SPLINE
SPL {X   -93.623, Y  +806.710, Z    +0.000, E1   -55.511, E3 +129906.770}
SPL {X  -138.493, Y  +759.115, Z    +0.000, E1   -50.023, E3 +129954.598}
SPL {X  -149.871, Y  +737.133, Z    +0.000, E1   -43.112, E3 +129960.012}
SPL {X  -157.876, Y  +713.320, Z    +0.000, E1   -31.448, E3 +129959.788}
SPL {X  -161.323, Y  +695.531, Z    +0.000, E1   -20.168, E3 +129961.831}
SPL {X  -162.626, Y  +681.447, Z    +0.000, E1    -9.120, E3 +129961.820}
SPL {X  -162.820, Y  +671.283, Z    +0.000, E1    +0.049, E3 +129961.332}
SPL {X  -162.820, Y  +665.565, Z    +0.000, E1   +11.206, E3 +129960.995}
SPL {X  -162.820, Y  +658.993, Z    +0.000, E1   +25.845, E3 +129961.066}
SPL {X  -162.820, Y  +652.443, Z    +0.000, E1   +38.206, E3 +129961.801}
SPL {X  -162.820, Y  +640.832, Z    +0.000, E1   +55.385, E3 +129960.515}
SPL {X  -162.820, Y  +625.562, Z    +0.000, E1   +67.658, E3 +129959.568}
SPL {X  -162.820, Y  +600.578, Z    +0.000, E1   +80.831, E3 +129951.166}
SPL {X  -162.820, Y  +567.495, Z    +0.000, E1   +70.620, E3 +129986.290}
SPL {X  -162.820, Y  +416.506, Z    +0.000, E1   +71.398, E3 +130070.636}
SPL {X  -162.820, Y  +411.010, Z    +0.000, E1   +70.614, E3 +130082.087}
SPL {X  -162.820, Y  +391.151, Z    +0.000, E1   +70.927, E3 +130093.542}
SPL {X  -159.025, Y  +345.550, Z    +0.000, E1   +73.389, E3 +130099.223}
SPL {X  -158.911, Y  +345.038, Z    +0.000, E1   +72.209, E3 +130111.381}
SPL {X  -157.738, Y  +340.137, Z    +0.000, E1   +71.006, E3 +130126.198}
SPL {X  -155.731, Y  +332.978, Z    +0.000, E1   +69.670, E3 +130142.847}
SPL {X  -154.241, Y  +328.346, Z    +0.000, E1   +68.710, E3 +130153.790}
SPL {X  -151.364, Y  +320.507, Z    +0.000, E1   +68.513, E3 +130161.416}
SPL {X  -147.865, Y  +312.336, Z    +0.000, E1   +67.945, E3 +130171.706}
SPL {X  -144.739, Y  +305.928, Z    +0.000, E1   +67.540, E3 +130179.290}
SPL {X  -141.308, Y  +299.614, Z    +0.000, E1   +67.079, E3 +130187.081}
SPL {X  -137.907, Y  +293.943, Z    +0.000, E1   +66.608, E3 +130194.059}
SPL {X  -134.802, Y  +289.183, Z    +0.000, E1   +66.143, E3 +130200.195}
SPL {X  -131.727, Y  +284.801, Z    +0.000, E1   +65.590, E3 +130206.210}
SPL {X  -128.890, Y  +281.012, Z    +0.000, E1   +65.392, E3 +130209.955}
SPL {X  -121.325, Y  +271.915, Z    +0.000, E1   +67.092, E3 +130209.521}
SPL {X   -79.997, Y  +238.687, Z    +0.000, E1   +54.340, E3 +130368.277}
ENDSPLINE

SPLINE
SPL {X  -139.099, Y  +295.872, Z    +0.000, E1   +47.860, E3 +130496.153}
SPL {X  -156.463, Y  +335.448, Z    +0.000, E1   +33.333, E3 +130506.861}
SPL {X  -161.312, Y  +358.394, Z    +0.000, E1   +19.478, E3 +130508.495}
SPL {X  -162.549, Y  +371.111, Z    +0.000, E1    +9.905, E3 +130508.555}
SPL {X  -162.818, Y  +379.769, Z    +0.000, E1    +2.607, E3 +130508.297}
SPL {X  -162.820, Y  +382.897, Z    +0.000, E1    -0.379, E3 +130507.781}
SPL {X  -162.820, Y  +387.689, Z    +0.000, E1    -9.147, E3 +130507.501}
SPL {X  -162.820, Y  +392.805, Z    +0.000, E1   -19.930, E3 +130507.474}
SPL {X  -162.820, Y  +397.742, Z    +0.000, E1   -30.068, E3 +130507.506}
SPL {X  -162.820, Y  +403.938, Z    +0.000, E1   -41.112, E3 +130507.486}
SPL {X  -162.820, Y  +415.430, Z    +0.000, E1   -55.307, E3 +130507.685}
SPL {X  -162.820, Y  +466.986, Z    +0.000, E1   -71.397, E3 +130519.444}
SPL {X  -162.820, Y  +661.594, Z    +0.000, E1   -73.988, E3 +130605.070}
ENDSPLINE

SPLINE
SPL {X  -162.820, Y  +634.363, Z    +0.000, E1   -70.793, E3 +130618.648}
ENDSPLINE

SPLINE
SPL {X  -162.820, Y  +649.777, Z    +0.000, E1   -70.953, E3 +130628.407}
SPL {X  -162.820, Y  +667.477, Z    +0.000, E1   -70.889, E3 +130641.716}
SPL {X  -162.462, Y  +684.286, Z    +0.000, E1   -70.880, E3 +130653.949}
SPL {X  -160.799, Y  +699.074, Z    +0.000, E1   -70.750, E3 +130665.813}
SPL {X  -158.733, Y  +709.754, Z    +0.000, E1   -70.504, E3 +130675.696}
SPL {X  -156.566, Y  +718.194, Z    +0.000, E1   -70.115, E3 +130685.177}
SPL {X  -153.268, Y  +728.449, Z    +0.000, E1   -69.855, E3 +130694.803}
SPL {X  -149.282, Y  +738.502, Z    +0.000, E1   -69.318, E3 +130706.323}
SPL {X  -145.460, Y  +746.655, Z    +0.000, E1   -68.995, E3 +130714.338}
SPL {X  -143.061, Y  +751.243, Z    +0.000, E1   -68.459, E3 +130721.332}
SPL {X  -139.143, Y  +758.055, Z    +0.000, E1   -68.038, E3 +130728.895}
SPL {X  -136.095, Y  +762.879, Z    +0.000, E1   -67.470, E3 +130735.529}
SPL {X  -133.055, Y  +767.344, Z    +0.000, E1   -67.024, E3 +130741.161}
SPL {X  -129.955, Y  +771.593, Z    +0.000, E1   -66.476, E3 +130746.802}
SPL {X  -125.283, Y  +777.493, Z    +0.000, E1   -66.879, E3 +130749.226}
SPL {X   -78.323, Y  +816.244, Z    +0.000, E1   -56.979, E3 +130856.322}
ENDSPLINE

SPLINE
SPL {X   -93.623, Y  +806.710, Z    +0.000, E1   -55.511, E3 +131002.008}
SPL {X  -138.493, Y  +759.115, Z    +0.000, E1   -50.023, E3 +131049.836}
SPL {X  -149.871, Y  +737.133, Z    +0.000, E1   -43.112, E3 +131055.250}
SPL {X  -157.876, Y  +713.320, Z    +0.000, E1   -31.448, E3 +131055.026}
SPL {X  -161.323, Y  +695.531, Z    +0.000, E1   -20.168, E3 +131057.069}
SPL {X  -162.626, Y  +681.447, Z    +0.000, E1    -9.120, E3 +131057.058}
SPL {X  -162.820, Y  +673.597, Z    +0.000, E1    -2.055, E3 +131057.052}
SPL {X  -162.820, Y  +671.476, Z    +0.000, E1    +0.020, E3 +131056.594}
SPL {X  -162.820, Y  +668.959, Z    +0.000, E1    +4.387, E3 +131056.315}
SPL {X  -162.820, Y  +664.344, Z    +0.000, E1   +14.120, E3 +131056.214}
SPL {X  -162.820, Y  +658.993, Z    +0.000, E1   +25.845, E3 +131056.304}
SPL {X  -162.820, Y  +652.443, Z    +0.000, E1   +38.206, E3 +131057.039}
SPL {X  -162.820, Y  +640.832, Z    +0.000, E1   +55.385, E3 +131055.753}
SPL {X  -162.820, Y  +617.334, Z    +0.000, E1   +73.158, E3 +131052.067}
SPL {X  -162.820, Y  +567.495, Z    +0.000, E1   +70.620, E3 +131081.528}
SPL {X  -162.820, Y  +416.506, Z    +0.000, E1   +71.398, E3 +131165.874}
SPL {X  -162.820, Y  +411.010, Z    +0.000, E1   +70.614, E3 +131177.325}
SPL {X  -162.820, Y  +399.588, Z    +0.000, E1   +70.462, E3 +131187.099}
SPL {X  -159.703, Y  +348.793, Z    +0.000, E1   +73.194, E3 +131194.403}
SPL {X  -158.809, Y  +344.584, Z    +0.000, E1   +72.042, E3 +131208.707}
SPL {X  -157.517, Y  +339.284, Z    +0.000, E1   +70.832, E3 +131223.408}
SPL {X  -155.731, Y  +332.978, Z    +0.000, E1   +69.670, E3 +131238.086}
SPL {X  -154.241, Y  +328.346, Z    +0.000, E1   +68.710, E3 +131249.028}
SPL {X  -151.364, Y  +320.507, Z    +0.000, E1   +68.513, E3 +131256.655}
SPL {X  -147.865, Y  +312.336, Z    +0.000, E1   +67.945, E3 +131266.944}
SPL {X  -144.739, Y  +305.928, Z    +0.000, E1   +67.540, E3 +131274.528}
SPL {X  -141.308, Y  +299.614, Z    +0.000, E1   +67.079, E3 +131282.319}
SPL {X  -137.907, Y  +293.943, Z    +0.000, E1   +66.608, E3 +131289.297}
SPL {X  -134.802, Y  +289.183, Z    +0.000, E1   +66.143, E3 +131295.433}
SPL {X  -131.727, Y  +284.801, Z    +0.000, E1   +65.590, E3 +131301.448}
SPL {X  -128.890, Y  +281.012, Z    +0.000, E1   +65.392, E3 +131305.193}
SPL {X  -121.325, Y  +271.915, Z    +0.000, E1   +67.092, E3 +131304.759}
SPL {X   -79.997, Y  +238.687, Z    +0.000, E1   +54.340, E3 +131463.515}
ENDSPLINE

SPLINE
SPL {X  -139.099, Y  +295.872, Z    +0.000, E1   +47.860, E3 +131591.391}
SPL {X  -153.884, Y  +327.303, Z    +0.000, E1   +37.422, E3 +131602.618}
SPL {X  -160.677, Y  +354.168, Z    +0.000, E1   +22.396, E3 +131603.144}
SPL {X  -162.549, Y  +371.111, Z    +0.000, E1    +9.905, E3 +131603.793}
SPL {X  -162.818, Y  +379.769, Z    +0.000, E1    +2.607, E3 +131603.535}
SPL {X  -162.820, Y  +382.500, Z    +0.000, E1    +0.000, E3 +131603.105}
SPL {X  -162.820, Y  +384.989, Z    +0.000, E1    -3.865, E3 +131602.832}
SPL {X  -162.820, Y  +391.404, Z    +0.000, E1   -16.767, E3 +131602.678}
SPL {X  -162.820, Y  +397.742, Z    +0.000, E1   -30.068, E3 +131602.744}
SPL {X  -162.820, Y  +403.938, Z    +0.000, E1   -41.112, E3 +131602.724}
SPL {X  -162.820, Y  +415.430, Z    +0.000, E1   -55.307, E3 +131602.923}
SPL {X  -162.820, Y  +466.986, Z    +0.000, E1   -71.397, E3 +131614.682}
SPL {X  -162.820, Y  +661.594, Z    +0.000, E1   -73.988, E3 +131700.309}
ENDSPLINE

SPLINE
SPL {X  -162.820, Y  +634.363, Z    +0.000, E1   -70.793, E3 +131713.886}
ENDSPLINE

SPLINE
SPL {X  -162.820, Y  +649.777, Z    +0.000, E1   -70.953, E3 +131723.645}
SPL {X  -162.820, Y  +667.477, Z    +0.000, E1   -70.889, E3 +131736.954}
SPL {X  -162.462, Y  +684.286, Z    +0.000, E1   -70.880, E3 +131749.187}
SPL {X  -160.799, Y  +699.074, Z    +0.000, E1   -70.750, E3 +131761.051}
SPL {X  -158.733, Y  +709.754, Z    +0.000, E1   -70.504, E3 +131770.934}
SPL {X  -156.566, Y  +718.194, Z    +0.000, E1   -70.115, E3 +131780.415}
SPL {X  -153.268, Y  +728.449, Z    +0.000, E1   -69.855, E3 +131790.041}
SPL {X  -150.033, Y  +736.750, Z    +0.000, E1   -69.498, E3 +131798.752}
SPL {X  -146.704, Y  +744.128, Z    +0.000, E1   -68.985, E3 +131807.875}
SPL {X  -143.061, Y  +751.243, Z    +0.000, E1   -68.459, E3 +131816.570}
SPL {X  -139.143, Y  +758.055, Z    +0.000, E1   -68.038, E3 +131824.133}
SPL {X  -136.095, Y  +762.879, Z    +0.000, E1   -67.470, E3 +131830.767}
SPL {X  -133.055, Y  +767.344, Z    +0.000, E1   -67.024, E3 +131836.399}
SPL {X  -129.955, Y  +771.593, Z    +0.000, E1   -66.476, E3 +131842.040}
SPL {X  -125.283, Y  +777.493, Z    +0.000, E1   -66.879, E3 +131844.464}
SPL {X   -78.323, Y  +816.244, Z    +0.000, E1   -56.979, E3 +131951.560}
ENDSPLINE

SPLINE
SPL {X   -93.623, Y  +806.710, Z    +0.000, E1   -55.511, E3 +132097.246}
SPL {X  -143.027, Y  +751.304, Z    +0.000, E1   -47.932, E3 +132147.307}
SPL {X  -157.876, Y  +713.320, Z    +0.000, E1   -31.448, E3 +132150.264}
SPL {X  -161.323, Y  +695.531, Z    +0.000, E1   -20.168, E3 +132152.308}
SPL {X  -162.428, Y  +684.786, Z    +0.000, E1   -11.829, E3 +132152.205}
SPL {X  -162.809, Y  +675.372, Z    +0.000, E1    -3.788, E3 +132152.319}
SPL {X  -162.820, Y  +671.476, Z    +0.000, E1    +0.020, E3 +132151.832}
SPL {X  -162.820, Y  +668.959, Z    +0.000, E1    +4.387, E3 +132151.553}
SPL {X  -162.820, Y  +664.344, Z    +0.000, E1   +14.120, E3 +132151.452}
SPL {X  -162.820, Y  +658.993, Z    +0.000, E1   +25.845, E3 +132151.542}
SPL {X  -162.820, Y  +652.443, Z    +0.000, E1   +38.206, E3 +132152.277}
SPL {X  -162.820, Y  +640.832, Z    +0.000, E1   +55.385, E3 +132150.991}
SPL {X  -162.820, Y  +625.562, Z    +0.000, E1   +67.658, E3 +132150.044}
SPL {X  -162.820, Y  +600.578, Z    +0.000, E1   +80.831, E3 +132141.642}
SPL {X  -162.820, Y  +567.495, Z    +0.000, E1   +70.620, E3 +132176.767}
SPL {X  -162.820, Y  +416.506, Z    +0.000, E1   +71.398, E3 +132261.112}
SPL {X  -162.820, Y  +411.010, Z    +0.000, E1   +70.614, E3 +132272.563}
SPL {X  -162.820, Y  +399.588, Z    +0.000, E1   +70.462, E3 +132282.337}
SPL {X  -159.703, Y  +348.793, Z    +0.000, E1   +73.194, E3 +132289.641}
SPL {X  -158.809, Y  +344.584, Z    +0.000, E1   +72.042, E3 +132303.946}
SPL {X  -157.517, Y  +339.284, Z    +0.000, E1   +70.832, E3 +132318.647}
SPL {X  -155.731, Y  +332.978, Z    +0.000, E1   +69.670, E3 +132333.324}
SPL {X  -153.052, Y  +324.954, Z    +0.000, E1   +68.671, E3 +132347.286}
SPL {X  -149.405, Y  +315.782, Z    +0.000, E1   +68.161, E3 +132358.052}
SPL {X  -145.408, Y  +307.240, Z    +0.000, E1   +67.667, E3 +132368.030}
SPL {X  -142.385, Y  +301.526, Z    +0.000, E1   +67.199, E3 +132375.262}
SPL {X  -138.888, Y  +295.526, Z    +0.000, E1   +66.767, E3 +132382.547}
SPL {X  -134.802, Y  +289.183, Z    +0.000, E1   +66.143, E3 +132390.671}
SPL {X  -131.727, Y  +284.801, Z    +0.000, E1   +65.590, E3 +132396.686}
SPL {X  -128.890, Y  +281.012, Z    +0.000, E1   +65.392, E3 +132400.431}
SPL {X  -121.325, Y  +271.915, Z    +0.000, E1   +67.092, E3 +132399.997}
SPL {X   -79.997, Y  +238.687, Z    +0.000, E1   +54.340, E3 +132558.753}
ENDSPLINE

SPLINE
SPL {X  -139.099, Y  +295.872, Z    +0.000, E1   +47.860, E3 +132686.629}
SPL {X  -156.463, Y  +335.448, Z    +0.000, E1   +33.333, E3 +132697.337}
SPL {X  -161.312, Y  +358.394, Z    +0.000, E1   +19.478, E3 +132698.972}
SPL {X  -162.549, Y  +371.111, Z    +0.000, E1    +9.905, E3 +132699.031}
SPL {X  -162.818, Y  +379.769, Z    +0.000, E1    +2.607, E3 +132698.773}
SPL {X  -162.820, Y  +382.897, Z    +0.000, E1    -0.379, E3 +132698.258}
SPL {X  -162.820, Y  +387.689, Z    +0.000, E1    -9.147, E3 +132697.977}
SPL {X  -162.820, Y  +392.805, Z    +0.000, E1   -19.930, E3 +132697.950}
SPL {X  -162.820, Y  +397.742, Z    +0.000, E1   -30.068, E3 +132697.982}
SPL {X  -162.820, Y  +403.938, Z    +0.000, E1   -41.112, E3 +132697.962}
SPL {X  -162.820, Y  +415.430, Z    +0.000, E1   -55.307, E3 +132698.161}
SPL {X  -162.820, Y  +466.986, Z    +0.000, E1   -71.397, E3 +132709.920}
SPL {X  -162.820, Y  +661.594, Z    +0.000, E1   -73.988, E3 +132795.547}
ENDSPLINE

SPLINE
SPL {X  -162.820, Y  +639.523, Z    +0.000, E1   -70.828, E3 +132812.623}
ENDSPLINE

SPLINE
SPL {X  -162.820, Y  +655.227, Z    +0.000, E1   -71.020, E3 +132822.049}
SPL {X  -162.820, Y  +667.477, Z    +0.000, E1   -70.889, E3 +132832.192}
SPL {X  -162.097, Y  +688.831, Z    +0.000, E1   -70.910, E3 +132847.563}
SPL {X  -159.319, Y  +707.081, Z    +0.000, E1   -70.563, E3 +132863.849}
SPL {X  -155.769, Y  +720.894, Z    +0.000, E1   -70.077, E3 +132878.059}
SPL {X  -150.995, Y  +734.417, Z    +0.000, E1   -69.635, E3 +132891.436}
SPL {X  -146.704, Y  +744.128, Z    +0.000, E1   -68.985, E3 +132903.113}
SPL {X  -143.061, Y  +751.243, Z    +0.000, E1   -68.459, E3 +132911.808}
SPL {X  -139.143, Y  +758.055, Z    +0.000, E1   -68.038, E3 +132919.371}
SPL {X  -136.095, Y  +762.879, Z    +0.000, E1   -67.470, E3 +132926.006}
SPL {X  -133.055, Y  +767.344, Z    +0.000, E1   -67.024, E3 +132931.637}
SPL {X  -129.955, Y  +771.593, Z    +0.000, E1   -66.476, E3 +132937.278}
SPL {X  -125.283, Y  +777.493, Z    +0.000, E1   -66.879, E3 +132939.702}
SPL {X   -78.323, Y  +816.244, Z    +0.000, E1   -56.979, E3 +133046.798}
ENDSPLINE

SPLINE
SPL {X   -93.623, Y  +806.710, Z    +0.000, E1   -55.511, E3 +133192.484}
SPL {X  -143.027, Y  +751.304, Z    +0.000, E1   -47.932, E3 +133242.545}
SPL {X  -157.876, Y  +713.320, Z    +0.000, E1   -31.448, E3 +133245.502}
SPL {X  -161.323, Y  +695.531, Z    +0.000, E1   -20.168, E3 +133247.546}
SPL {X  -162.428, Y  +684.786, Z    +0.000, E1   -11.829, E3 +133247.443}
SPL {X  -162.809, Y  +675.372, Z    +0.000, E1    -3.788, E3 +133247.557}
SPL {X  -162.820, Y  +671.476, Z    +0.000, E1    +0.020, E3 +133247.070}
SPL {X  -162.820, Y  +668.959, Z    +0.000, E1    +4.387, E3 +133246.791}
SPL {X  -162.820, Y  +664.344, Z    +0.000, E1   +14.120, E3 +133246.690}
SPL {X  -162.820, Y  +658.993, Z    +0.000, E1   +25.845, E3 +133246.780}
SPL {X  -162.820, Y  +652.443, Z    +0.000, E1   +38.206, E3 +133247.515}
SPL {X  -162.820, Y  +640.832, Z    +0.000, E1   +55.385, E3 +133246.229}
SPL {X  -162.820, Y  +617.334, Z    +0.000, E1   +73.158, E3 +133242.543}
SPL {X  -162.820, Y  +567.495, Z    +0.000, E1   +70.620, E3 +133272.005}
SPL {X  -162.820, Y  +416.506, Z    +0.000, E1   +71.398, E3 +133356.350}
SPL {X  -162.820, Y  +411.010, Z    +0.000, E1   +70.614, E3 +133367.801}
SPL {X  -162.820, Y  +391.151, Z    +0.000, E1   +70.927, E3 +133379.256}
SPL {X  -159.025, Y  +345.550, Z    +0.000, E1   +73.389, E3 +133384.937}
ENDSPLINE

SPLINE
SPL {X  -159.121, Y  +345.992, Z    +0.000, E1   +72.455, E3 +133393.904}
ENDSPLINE

SPLINE
SPL {X  -158.667, Y  +343.959, Z    +0.000, E1   +71.763, E3 +133402.012}
SPL {X  -157.517, Y  +339.284, Z    +0.000, E1   +70.832, E3 +133413.885}
SPL {X  -155.731, Y  +332.978, Z    +0.000, E1   +69.670, E3 +133428.562}
SPL {X  -154.241, Y  +328.346, Z    +0.000, E1   +68.710, E3 +133439.505}
SPL {X  -151.364, Y  +320.507, Z    +0.000, E1   +68.513, E3 +133447.131}
SPL {X  -147.865, Y  +312.336, Z    +0.000, E1   +67.945, E3 +133457.421}
SPL {X  -143.686, Y  +303.920, Z    +0.000, E1   +67.419, E3 +133467.451}
SPL {X  -138.888, Y  +295.526, Z    +0.000, E1   +66.767, E3 +133477.785}
SPL {X  -134.802, Y  +289.183, Z    +0.000, E1   +66.143, E3 +133485.909}
SPL {X  -131.727, Y  +284.801, Z    +0.000, E1   +65.590, E3 +133491.924}
SPL {X  -128.890, Y  +281.012, Z    +0.000, E1   +65.392, E3 +133495.669}
SPL {X  -121.325, Y  +271.915, Z    +0.000, E1   +67.092, E3 +133495.235}
SPL {X   -79.997, Y  +238.687, Z    +0.000, E1   +54.340, E3 +133653.991}
ENDSPLINE

SPLINE
SPL {X  -139.099, Y  +295.872, Z    +0.000, E1   +47.860, E3 +133781.867}
SPL {X  -156.463, Y  +335.448, Z    +0.000, E1   +33.333, E3 +133792.575}
SPL {X  -161.312, Y  +358.394, Z    +0.000, E1   +19.478, E3 +133794.210}
SPL {X  -162.549, Y  +371.111, Z    +0.000, E1    +9.905, E3 +133794.270}
SPL {X  -162.818, Y  +379.769, Z    +0.000, E1    +2.607, E3 +133794.012}
SPL {X  -162.820, Y  +382.897, Z    +0.000, E1    -0.379, E3 +133793.496}
SPL {X  -162.820, Y  +387.689, Z    +0.000, E1    -9.147, E3 +133793.215}
SPL {X  -162.820, Y  +392.805, Z    +0.000, E1   -19.930, E3 +133793.188}
SPL {X  -162.820, Y  +397.742, Z    +0.000, E1   -30.068, E3 +133793.221}
SPL {X  -162.820, Y  +403.938, Z    +0.000, E1   -41.112, E3 +133793.200}
SPL {X  -162.820, Y  +415.430, Z    +0.000, E1   -55.307, E3 +133793.399}
SPL {X  -162.820, Y  +466.986, Z    +0.000, E1   -71.397, E3 +133805.158}
SPL {X  -162.820, Y  +661.594, Z    +0.000, E1   -73.988, E3 +133890.785}
ENDSPLINE

SPLINE
SPL {X  -162.820, Y  +634.363, Z    +0.000, E1   -70.793, E3 +133904.363}
ENDSPLINE

SPLINE
SPL {X  -162.820, Y  +649.777, Z    +0.000, E1   -70.953, E3 +133914.121}
SPL {X  -162.820, Y  +667.477, Z    +0.000, E1   -70.889, E3 +133927.430}
SPL {X  -162.462, Y  +684.286, Z    +0.000, E1   -70.880, E3 +133939.663}
SPL {X  -160.799, Y  +699.074, Z    +0.000, E1   -70.750, E3 +133951.528}
SPL {X  -158.733, Y  +709.754, Z    +0.000, E1   -70.504, E3 +133961.410}
SPL {X  -156.566, Y  +718.194, Z    +0.000, E1   -70.115, E3 +133970.892}
SPL {X  -153.268, Y  +728.449, Z    +0.000, E1   -69.855, E3 +133980.517}
SPL {X  -150.033, Y  +736.750, Z    +0.000, E1   -69.498, E3 +133989.229}
SPL {X  -146.704, Y  +744.128, Z    +0.000, E1   -68.985, E3 +133998.351}
SPL {X  -143.061, Y  +751.243, Z    +0.000, E1   -68.459, E3 +134007.046}
SPL {X  -139.143, Y  +758.055, Z    +0.000, E1   -68.038, E3 +134014.609}
SPL {X  -136.095, Y  +762.879, Z    +0.000, E1   -67.470, E3 +134021.244}
SPL {X  -133.055, Y  +767.344, Z    +0.000, E1   -67.024, E3 +134026.875}
SPL {X  -129.955, Y  +771.593, Z    +0.000, E1   -66.476, E3 +134032.516}
SPL {X  -125.283, Y  +777.493, Z    +0.000, E1   -66.879, E3 +134034.941}
SPL {X   -78.323, Y  +816.244, Z    +0.000, E1   -56.979, E3 +134142.036}
ENDSPLINE

SPLINE
SPL {X   -93.623, Y  +806.710, Z    +0.000, E1   -55.511, E3 +134287.722}
SPL {X  -143.027, Y  +751.304, Z    +0.000, E1   -47.932, E3 +134337.783}
SPL {X  -157.876, Y  +713.320, Z    +0.000, E1   -31.448, E3 +134340.740}
SPL {X  -161.323, Y  +695.531, Z    +0.000, E1   -20.168, E3 +134342.784}
SPL {X  -162.428, Y  +684.786, Z    +0.000, E1   -11.829, E3 +134342.681}
SPL {X  -162.809, Y  +675.372, Z    +0.000, E1    -3.788, E3 +134342.795}
SPL {X  -162.820, Y  +671.476, Z    +0.000, E1    +0.020, E3 +134342.308}
SPL {X  -162.820, Y  +668.959, Z    +0.000, E1    +4.387, E3 +134342.029}
SPL {X  -162.820, Y  +664.344, Z    +0.000, E1   +14.120, E3 +134341.928}
SPL {X  -162.820, Y  +658.993, Z    +0.000, E1   +25.845, E3 +134342.018}
SPL {X  -162.820, Y  +652.443, Z    +0.000, E1   +38.206, E3 +134342.754}
SPL {X  -162.820, Y  +640.832, Z    +0.000, E1   +55.385, E3 +134341.467}
SPL {X  -162.820, Y  +625.562, Z    +0.000, E1   +67.658, E3 +134340.520}
SPL {X  -162.820, Y  +600.578, Z    +0.000, E1   +80.831, E3 +134332.118}
SPL {X  -162.820, Y  +567.495, Z    +0.000, E1   +70.620, E3 +134367.243}
SPL {X  -162.820, Y  +416.506, Z    +0.000, E1   +71.398, E3 +134451.588}
SPL {X  -162.820, Y  +411.010, Z    +0.000, E1   +70.614, E3 +134463.039}
SPL {X  -162.820, Y  +399.588, Z    +0.000, E1   +70.462, E3 +134472.813}
SPL {X  -159.703, Y  +348.793, Z    +0.000, E1   +73.194, E3 +134480.117}
SPL {X  -158.809, Y  +344.584, Z    +0.000, E1   +72.042, E3 +134494.422}
SPL {X  -157.517, Y  +339.284, Z    +0.000, E1   +70.832, E3 +134509.123}
SPL {X  -155.731, Y  +332.978, Z    +0.000, E1   +69.670, E3 +134523.800}
SPL {X  -153.052, Y  +324.954, Z    +0.000, E1   +68.671, E3 +134537.762}
SPL {X  -149.405, Y  +315.782, Z    +0.000, E1   +68.161, E3 +134548.528}
SPL {X  -145.408, Y  +307.240, Z    +0.000, E1   +67.667, E3 +134558.506}
SPL {X  -142.385, Y  +301.526, Z    +0.000, E1   +67.199, E3 +134565.738}
SPL {X  -138.888, Y  +295.526, Z    +0.000, E1   +66.767, E3 +134573.024}
SPL {X  -134.802, Y  +289.183, Z    +0.000, E1   +66.143, E3 +134581.148}
SPL {X  -131.727, Y  +284.801, Z    +0.000, E1   +65.590, E3 +134587.162}
SPL {X  -128.890, Y  +281.012, Z    +0.000, E1   +65.392, E3 +134590.907}
SPL {X  -121.325, Y  +271.915, Z    +0.000, E1   +67.092, E3 +134590.473}
SPL {X   -79.997, Y  +238.687, Z    +0.000, E1   +54.340, E3 +134749.229}
ENDSPLINE

SPLINE
SPL {X  -139.099, Y  +295.872, Z    +0.000, E1   +47.860, E3 +134877.105}
SPL {X  -156.463, Y  +335.448, Z    +0.000, E1   +33.333, E3 +134887.813}
SPL {X  -161.312, Y  +358.394, Z    +0.000, E1   +19.478, E3 +134889.448}
SPL {X  -162.549, Y  +371.111, Z    +0.000, E1    +9.905, E3 +134889.508}
SPL {X  -162.818, Y  +379.769, Z    +0.000, E1    +2.607, E3 +134889.250}
SPL {X  -162.820, Y  +382.897, Z    +0.000, E1    -0.379, E3 +134888.734}
SPL {X  -162.820, Y  +387.689, Z    +0.000, E1    -9.147, E3 +134888.453}
SPL {X  -162.820, Y  +392.805, Z    +0.000, E1   -19.930, E3 +134888.426}
SPL {X  -162.820, Y  +397.742, Z    +0.000, E1   -30.068, E3 +134888.459}
SPL {X  -162.820, Y  +403.938, Z    +0.000, E1   -41.112, E3 +134888.438}
SPL {X  -162.820, Y  +415.430, Z    +0.000, E1   -55.307, E3 +134888.637}
SPL {X  -162.820, Y  +466.986, Z    +0.000, E1   -71.397, E3 +134900.397}
SPL {X  -162.820, Y  +661.594, Z    +0.000, E1   -73.988, E3 +134986.023}
ENDSPLINE

SPLINE
SPL {X  -162.820, Y  +639.523, Z    +0.000, E1   -70.828, E3 +135003.099}
ENDSPLINE

SPLINE
SPL {X  -162.820, Y  +655.227, Z    +0.000, E1   -71.020, E3 +135012.525}
SPL {X  -162.820, Y  +667.477, Z    +0.000, E1   -70.889, E3 +135022.668}
SPL {X  -162.097, Y  +688.831, Z    +0.000, E1   -70.910, E3 +135038.039}
SPL {X  -159.319, Y  +707.081, Z    +0.000, E1   -70.563, E3 +135054.325}
SPL {X  -155.769, Y  +720.894, Z    +0.000, E1   -70.077, E3 +135068.536}
SPL {X  -150.995, Y  +734.417, Z    +0.000, E1   -69.635, E3 +135081.912}
SPL {X  -146.704, Y  +744.128, Z    +0.000, E1   -68.985, E3 +135093.589}
SPL {X  -143.061, Y  +751.243, Z    +0.000, E1   -68.459, E3 +135102.284}
SPL {X  -139.143, Y  +758.055, Z    +0.000, E1   -68.038, E3 +135109.847}
SPL {X  -136.095, Y  +762.879, Z    +0.000, E1   -67.470, E3 +135116.482}
SPL {X  -133.055, Y  +767.344, Z    +0.000, E1   -67.024, E3 +135122.113}
SPL {X  -129.955, Y  +771.593, Z    +0.000, E1   -66.476, E3 +135127.754}
SPL {X  -125.283, Y  +777.493, Z    +0.000, E1   -66.879, E3 +135130.179}
SPL {X   -78.323, Y  +816.244, Z    +0.000, E1   -56.979, E3 +135237.274}
ENDSPLINE

SPLINE
SPL {X   -93.623, Y  +806.710, Z    +0.000, E1   -55.511, E3 +135382.960}
SPL {X  -143.027, Y  +751.304, Z    +0.000, E1   -47.932, E3 +135433.021}
SPL {X  -157.876, Y  +713.320, Z    +0.000, E1   -31.448, E3 +135435.978}
SPL {X  -161.323, Y  +695.531, Z    +0.000, E1   -20.168, E3 +135438.022}
SPL {X  -162.428, Y  +684.786, Z    +0.000, E1   -11.829, E3 +135437.919}
SPL {X  -162.809, Y  +675.372, Z    +0.000, E1    -3.788, E3 +135438.033}
SPL {X  -162.820, Y  +671.476, Z    +0.000, E1    +0.020, E3 +135437.546}
SPL {X  -162.820, Y  +668.959, Z    +0.000, E1    +4.387, E3 +135437.267}
SPL {X  -162.820, Y  +664.344, Z    +0.000, E1   +14.120, E3 +135437.166}
SPL {X  -162.820, Y  +658.993, Z    +0.000, E1   +25.845, E3 +135437.256}
SPL {X  -162.820, Y  +652.443, Z    +0.000, E1   +38.206, E3 +135437.992}
SPL {X  -162.820, Y  +640.832, Z    +0.000, E1   +55.385, E3 +135436.705}
SPL {X  -162.820, Y  +617.334, Z    +0.000, E1   +73.158, E3 +135433.019}
SPL {X  -162.820, Y  +567.495, Z    +0.000, E1   +70.620, E3 +135462.481}
SPL {X  -162.820, Y  +416.506, Z    +0.000, E1   +71.398, E3 +135546.826}
SPL {X  -162.820, Y  +411.010, Z    +0.000, E1   +70.614, E3 +135558.278}
SPL {X  -162.820, Y  +391.151, Z    +0.000, E1   +70.927, E3 +135569.732}
SPL {X  -159.025, Y  +345.550, Z    +0.000, E1   +73.389, E3 +135575.413}
ENDSPLINE

SPLINE
SPL {X  -159.121, Y  +345.992, Z    +0.000, E1   +72.455, E3 +135584.380}
ENDSPLINE

SPLINE
SPL {X  -158.667, Y  +343.959, Z    +0.000, E1   +71.763, E3 +135592.488}
SPL {X  -157.517, Y  +339.284, Z    +0.000, E1   +70.832, E3 +135604.361}
SPL {X  -155.731, Y  +332.978, Z    +0.000, E1   +69.670, E3 +135619.038}
SPL {X  -153.052, Y  +324.954, Z    +0.000, E1   +68.671, E3 +135633.001}
SPL {X  -148.581, Y  +313.911, Z    +0.000, E1   +68.095, E3 +135645.791}
SPL {X  -143.686, Y  +303.920, Z    +0.000, E1   +67.419, E3 +135657.927}
SPL {X  -138.888, Y  +295.526, Z    +0.000, E1   +66.767, E3 +135668.262}
SPL {X  -134.802, Y  +289.183, Z    +0.000, E1   +66.143, E3 +135676.386}
SPL {X  -131.727, Y  +284.801, Z    +0.000, E1   +65.590, E3 +135682.400}
SPL {X  -128.890, Y  +281.012, Z    +0.000, E1   +65.392, E3 +135686.145}
SPL {X  -121.325, Y  +271.915, Z    +0.000, E1   +67.092, E3 +135685.711}
SPL {X   -79.997, Y  +238.687, Z    +0.000, E1   +54.340, E3 +135844.468}
ENDSPLINE

SPLINE
SPL {X  -139.099, Y  +295.872, Z    +0.000, E1   +47.860, E3 +135972.343}
SPL {X  -156.463, Y  +335.448, Z    +0.000, E1   +33.333, E3 +135983.051}
SPL {X  -161.312, Y  +358.394, Z    +0.000, E1   +19.478, E3 +135984.686}
SPL {X  -162.549, Y  +371.111, Z    +0.000, E1    +9.905, E3 +135984.746}
SPL {X  -162.818, Y  +379.769, Z    +0.000, E1    +2.607, E3 +135984.488}
SPL {X  -162.820, Y  +382.897, Z    +0.000, E1    -0.379, E3 +135983.972}
SPL {X  -162.820, Y  +387.689, Z    +0.000, E1    -9.147, E3 +135983.691}
SPL {X  -162.820, Y  +392.805, Z    +0.000, E1   -19.930, E3 +135983.664}
SPL {X  -162.820, Y  +397.742, Z    +0.000, E1   -30.068, E3 +135983.697}
SPL {X  -162.820, Y  +403.938, Z    +0.000, E1   -41.112, E3 +135983.676}
SPL {X  -162.820, Y  +415.430, Z    +0.000, E1   -55.307, E3 +135983.875}
SPL {X  -162.820, Y  +466.986, Z    +0.000, E1   -71.397, E3 +135995.635}
SPL {X  -162.820, Y  +661.594, Z    +0.000, E1   -73.988, E3 +136081.261}
ENDSPLINE

SPLINE
SPL {X  -162.820, Y  +639.523, Z    +0.000, E1   -70.828, E3 +136098.338}
ENDSPLINE

SPLINE
SPL {X  -162.820, Y  +655.227, Z    +0.000, E1   -71.020, E3 +136107.763}
SPL {X  -162.820, Y  +667.477, Z    +0.000, E1   -70.889, E3 +136117.906}
SPL {X  -162.462, Y  +684.286, Z    +0.000, E1   -70.880, E3 +136130.139}
SPL {X  -160.799, Y  +699.074, Z    +0.000, E1   -70.750, E3 +136142.004}
SPL {X  -158.733, Y  +709.754, Z    +0.000, E1   -70.504, E3 +136151.886}
SPL {X  -156.566, Y  +718.194, Z    +0.000, E1   -70.115, E3 +136161.368}
SPL {X  -153.268, Y  +728.449, Z    +0.000, E1   -69.855, E3 +136170.993}
SPL {X  -149.282, Y  +738.502, Z    +0.000, E1   -69.318, E3 +136182.514}
SPL {X  -145.460, Y  +746.655, Z    +0.000, E1   -68.995, E3 +136190.528}
SPL {X  -143.061, Y  +751.243, Z    +0.000, E1   -68.459, E3 +136197.523}
SPL {X  -139.143, Y  +758.055, Z    +0.000, E1   -68.038, E3 +136205.085}
SPL {X  -136.095, Y  +762.879, Z    +0.000, E1   -67.470, E3 +136211.720}
SPL {X  -133.055, Y  +767.344, Z    +0.000, E1   -67.024, E3 +136217.351}
SPL {X  -129.955, Y  +771.593, Z    +0.000, E1   -66.476, E3 +136222.992}
SPL {X  -125.283, Y  +777.493, Z    +0.000, E1   -66.879, E3 +136225.417}
SPL {X   -78.323, Y  +816.244, Z    +0.000, E1   -56.979, E3 +136332.512}
ENDSPLINE

SPLINE
SPL {X   -93.623, Y  +806.710, Z    +0.000, E1   -55.511, E3 +136478.198}
SPL {X  -143.027, Y  +751.304, Z    +0.000, E1   -47.932, E3 +136528.259}
SPL {X  -157.876, Y  +713.320, Z    +0.000, E1   -31.448, E3 +136531.216}
SPL {X  -161.323, Y  +695.531, Z    +0.000, E1   -20.168, E3 +136533.260}
SPL {X  -162.428, Y  +684.786, Z    +0.000, E1   -11.829, E3 +136533.157}
SPL {X  -162.809, Y  +675.372, Z    +0.000, E1    -3.788, E3 +136533.271}
SPL {X  -162.820, Y  +671.476, Z    +0.000, E1    +0.020, E3 +136532.785}
SPL {X  -162.820, Y  +668.959, Z    +0.000, E1    +4.387, E3 +136532.505}
SPL {X  -162.820, Y  +664.344, Z    +0.000, E1   +14.120, E3 +136532.404}
SPL {X  -162.820, Y  +658.993, Z    +0.000, E1   +25.845, E3 +136532.494}
SPL {X  -162.820, Y  +652.443, Z    +0.000, E1   +38.206, E3 +136533.230}
SPL {X  -162.820, Y  +640.832, Z    +0.000, E1   +55.385, E3 +136531.943}
SPL {X  -162.820, Y  +625.562, Z    +0.000, E1   +67.658, E3 +136530.997}
SPL {X  -162.820, Y  +600.578, Z    +0.000, E1   +80.831, E3 +136522.594}
SPL {X  -162.820, Y  +567.495, Z    +0.000, E1   +70.620, E3 +136557.719}
SPL {X  -162.820, Y  +416.506, Z    +0.000, E1   +71.398, E3 +136642.065}
SPL {X  -162.820, Y  +411.010, Z    +0.000, E1   +70.614, E3 +136653.516}
SPL {X  -162.820, Y  +399.588, Z    +0.000, E1   +70.462, E3 +136663.289}
SPL {X  -159.703, Y  +348.793, Z    +0.000, E1   +73.194, E3 +136670.594}
SPL {X  -158.911, Y  +345.038, Z    +0.000, E1   +72.209, E3 +136682.810}
SPL {X  -157.738, Y  +340.137, Z    +0.000, E1   +71.006, E3 +136697.626}
SPL {X  -155.731, Y  +332.978, Z    +0.000, E1   +69.670, E3 +136714.276}
SPL {X  -153.052, Y  +324.954, Z    +0.000, E1   +68.671, E3 +136728.239}
SPL {X  -148.581, Y  +313.911, Z    +0.000, E1   +68.095, E3 +136741.029}
SPL {X  -143.686, Y  +303.920, Z    +0.000, E1   +67.419, E3 +136753.165}
SPL {X  -138.888, Y  +295.526, Z    +0.000, E1   +66.767, E3 +136763.500}
SPL {X  -134.802, Y  +289.183, Z    +0.000, E1   +66.143, E3 +136771.624}
SPL {X  -131.727, Y  +284.801, Z    +0.000, E1   +65.590, E3 +136777.638}
SPL {X  -128.890, Y  +281.012, Z    +0.000, E1   +65.392, E3 +136781.384}
SPL {X  -121.325, Y  +271.915, Z    +0.000, E1   +67.092, E3 +136780.949}
SPL {X   -79.997, Y  +238.687, Z    +0.000, E1   +54.340, E3 +136939.706}
ENDSPLINE

SPLINE
SPL {X  -139.099, Y  +295.872, Z    +0.000, E1   +47.860, E3 +137067.581}
SPL {X  -156.463, Y  +335.448, Z    +0.000, E1   +33.333, E3 +137078.289}
SPL {X  -161.312, Y  +358.394, Z    +0.000, E1   +19.478, E3 +137079.924}
SPL {X  -162.549, Y  +371.111, Z    +0.000, E1    +9.905, E3 +137079.984}
SPL {X  -162.818, Y  +379.769, Z    +0.000, E1    +2.607, E3 +137079.726}
SPL {X  -162.820, Y  +382.500, Z    +0.000, E1    +0.000, E3 +137079.295}
SPL {X  -162.820, Y  +384.989, Z    +0.000, E1    -3.865, E3 +137079.022}
SPL {X  -162.820, Y  +391.404, Z    +0.000, E1   -16.767, E3 +137078.869}
SPL {X  -162.820, Y  +397.742, Z    +0.000, E1   -30.068, E3 +137078.935}
SPL {X  -162.820, Y  +403.938, Z    +0.000, E1   -41.112, E3 +137078.914}
SPL {X  -162.820, Y  +415.430, Z    +0.000, E1   -55.307, E3 +137079.113}
SPL {X  -162.820, Y  +466.986, Z    +0.000, E1   -71.397, E3 +137090.873}
SPL {X  -162.820, Y  +661.594, Z    +0.000, E1   -73.988, E3 +137176.499}
ENDSPLINE

SPLINE
SPL {X  -162.820, Y  +634.363, Z    +0.000, E1   -70.793, E3 +137190.077}
ENDSPLINE

SPLINE
SPL {X  -162.820, Y  +649.777, Z    +0.000, E1   -70.953, E3 +137199.836}
SPL {X  -162.820, Y  +667.477, Z    +0.000, E1   -70.889, E3 +137213.144}
SPL {X  -162.097, Y  +688.831, Z    +0.000, E1   -70.910, E3 +137228.515}
SPL {X  -159.319, Y  +707.081, Z    +0.000, E1   -70.563, E3 +137244.801}
SPL {X  -156.566, Y  +718.194, Z    +0.000, E1   -70.115, E3 +137256.606}
SPL {X  -153.268, Y  +728.449, Z    +0.000, E1   -69.855, E3 +137266.231}
SPL {X  -150.033, Y  +736.750, Z    +0.000, E1   -69.498, E3 +137274.943}
SPL {X  -146.704, Y  +744.128, Z    +0.000, E1   -68.985, E3 +137284.065}
SPL {X  -142.102, Y  +752.982, Z    +0.000, E1   -68.357, E3 +137294.804}
SPL {X  -136.987, Y  +761.506, Z    +0.000, E1   -67.725, E3 +137304.688}
SPL {X  -133.055, Y  +767.344, Z    +0.000, E1   -67.024, E3 +137312.589}
SPL {X  -129.955, Y  +771.593, Z    +0.000, E1   -66.476, E3 +137318.230}
SPL {X  -125.283, Y  +777.493, Z    +0.000, E1   -66.879, E3 +137320.655}
SPL {X   -78.323, Y  +816.244, Z    +0.000, E1   -56.979, E3 +137427.750}
ENDSPLINE

SPLINE
SPL {X   -93.623, Y  +806.710, Z    +0.000, E1   -55.511, E3 +137573.437}
SPL {X  -138.493, Y  +759.115, Z    +0.000, E1   -50.023, E3 +137621.265}
SPL {X  -149.871, Y  +737.133, Z    +0.000, E1   -43.112, E3 +137626.679}
SPL {X  -157.876, Y  +713.320, Z    +0.000, E1   -31.448, E3 +137626.454}
SPL {X  -161.323, Y  +695.531, Z    +0.000, E1   -20.168, E3 +137628.498}
SPL {X  -162.626, Y  +681.447, Z    +0.000, E1    -9.120, E3 +137628.487}
SPL {X  -162.820, Y  +671.283, Z    +0.000, E1    +0.049, E3 +137627.999}
SPL {X  -162.820, Y  +665.565, Z    +0.000, E1   +11.206, E3 +137627.662}
SPL {X  -162.820, Y  +658.993, Z    +0.000, E1   +25.845, E3 +137627.732}
SPL {X  -162.820, Y  +650.479, Z    +0.000, E1   +41.861, E3 +137627.891}
SPL {X  -162.820, Y  +638.661, Z    +0.000, E1   +57.186, E3 +137627.593}
SPL {X  -162.820, Y  +617.334, Z    +0.000, E1   +73.158, E3 +137623.495}
SPL {X  -162.820, Y  +567.495, Z    +0.000, E1   +70.620, E3 +137652.957}
SPL {X  -162.820, Y  +406.037, Z    +0.000, E1   +72.667, E3 +137731.694}
ENDSPLINE

SPLINE
SPL {X  -162.820, Y  +414.365, Z    +0.000, E1   +70.598, E3 +137746.540}
ENDSPLINE

SPLINE
SPL {X  -162.820, Y  +399.588, Z    +0.000, E1   +70.462, E3 +137758.527}
SPL {X  -159.703, Y  +348.793, Z    +0.000, E1   +73.194, E3 +137765.832}
SPL {X  -159.121, Y  +345.992, Z    +0.000, E1   +72.455, E3 +137774.856}
SPL {X  -158.667, Y  +343.959, Z    +0.000, E1   +71.763, E3 +137782.964}
SPL {X  -157.517, Y  +339.284, Z    +0.000, E1   +70.832, E3 +137794.837}
SPL {X  -155.731, Y  +332.978, Z    +0.000, E1   +69.670, E3 +137809.514}
SPL {X  -154.241, Y  +328.346, Z    +0.000, E1   +68.710, E3 +137820.457}
SPL {X  -151.364, Y  +320.507, Z    +0.000, E1   +68.513, E3 +137828.083}
SPL {X  -147.865, Y  +312.336, Z    +0.000, E1   +67.945, E3 +137838.373}
SPL {X  -144.739, Y  +305.928, Z    +0.000, E1   +67.540, E3 +137845.956}
SPL {X  -141.308, Y  +299.614, Z    +0.000, E1   +67.079, E3 +137853.747}
SPL {X  -137.907, Y  +293.943, Z    +0.000, E1   +66.608, E3 +137860.726}
SPL {X  -134.802, Y  +289.183, Z    +0.000, E1   +66.143, E3 +137866.862}
SPL {X  -131.727, Y  +284.801, Z    +0.000, E1   +65.590, E3 +137872.876}
SPL {X  -128.890, Y  +281.012, Z    +0.000, E1   +65.392, E3 +137876.622}
SPL {X  -121.325, Y  +271.915, Z    +0.000, E1   +67.092, E3 +137876.187}
SPL {X   -79.997, Y  +238.687, Z    +0.000, E1   +54.340, E3 +138034.944}
ENDSPLINE

SPLINE
SPL {X  -139.099, Y  +295.872, Z    +0.000, E1   +47.860, E3 +138162.819}
SPL {X  -156.463, Y  +335.448, Z    +0.000, E1   +33.333, E3 +138173.527}
SPL {X  -161.312, Y  +358.394, Z    +0.000, E1   +19.478, E3 +138175.162}
SPL {X  -162.549, Y  +371.111, Z    +0.000, E1    +9.905, E3 +138175.222}
SPL {X  -162.818, Y  +379.769, Z    +0.000, E1    +2.607, E3 +138174.964}
SPL {X  -162.820, Y  +382.897, Z    +0.000, E1    -0.379, E3 +138174.448}
SPL {X  -162.820, Y  +387.689, Z    +0.000, E1    -9.147, E3 +138174.167}
SPL {X  -162.820, Y  +392.805, Z    +0.000, E1   -19.930, E3 +138174.140}
SPL {X  -162.820, Y  +397.742, Z    +0.000, E1   -30.068, E3 +138174.173}
SPL {X  -162.820, Y  +403.938, Z    +0.000, E1   -41.112, E3 +138174.152}
SPL {X  -162.820, Y  +415.430, Z    +0.000, E1   -55.307, E3 +138174.351}
SPL {X  -162.820, Y  +466.986, Z    +0.000, E1   -71.397, E3 +138186.111}
SPL {X  -162.820, Y  +661.594, Z    +0.000, E1   -73.988, E3 +138271.737}
ENDSPLINE

SPLINE
SPL {X  -162.820, Y  +634.363, Z    +0.000, E1   -70.793, E3 +138285.315}
ENDSPLINE

SPLINE
SPL {X  -162.820, Y  +649.777, Z    +0.000, E1   -70.953, E3 +138295.074}
SPL {X  -162.820, Y  +667.477, Z    +0.000, E1   -70.889, E3 +138308.383}
SPL {X  -162.097, Y  +688.831, Z    +0.000, E1   -70.910, E3 +138323.753}
SPL {X  -159.319, Y  +707.081, Z    +0.000, E1   -70.563, E3 +138340.040}
SPL {X  -156.566, Y  +718.194, Z    +0.000, E1   -70.115, E3 +138351.844}
SPL {X  -153.268, Y  +728.449, Z    +0.000, E1   -69.855, E3 +138361.469}
SPL {X  -150.033, Y  +736.750, Z    +0.000, E1   -69.498, E3 +138370.181}
SPL {X  -146.704, Y  +744.128, Z    +0.000, E1   -68.985, E3 +138379.303}
SPL {X  -142.102, Y  +752.982, Z    +0.000, E1   -68.357, E3 +138390.042}
SPL {X  -138.073, Y  +759.791, Z    +0.000, E1   -67.958, E3 +138397.211}
SPL {X  -134.977, Y  +764.558, Z    +0.000, E1   -67.353, E3 +138404.132}
SPL {X  -130.728, Y  +770.560, Z    +0.000, E1   -66.612, E3 +138412.168}
SPL {X  -125.283, Y  +777.493, Z    +0.000, E1   -66.879, E3 +138415.893}
SPL {X   -78.323, Y  +816.244, Z    +0.000, E1   -56.979, E3 +138522.988}
ENDSPLINE

SPLINE
SPL {X   -93.623, Y  +806.710, Z    +0.000, E1   -55.511, E3 +138668.675}
SPL {X  -143.027, Y  +751.304, Z    +0.000, E1   -47.932, E3 +138718.735}
SPL {X  -157.876, Y  +713.320, Z    +0.000, E1   -31.448, E3 +138721.692}
SPL {X  -161.323, Y  +695.531, Z    +0.000, E1   -20.168, E3 +138723.736}
SPL {X  -162.626, Y  +681.447, Z    +0.000, E1    -9.120, E3 +138723.725}
SPL {X  -162.820, Y  +671.283, Z    +0.000, E1    +0.049, E3 +138723.237}
SPL {X  -162.820, Y  +665.565, Z    +0.000, E1   +11.206, E3 +138722.900}
SPL {X  -162.820, Y  +658.993, Z    +0.000, E1   +25.845, E3 +138722.970}
SPL {X  -162.820, Y  +650.479, Z    +0.000, E1   +41.861, E3 +138723.130}
SPL {X  -162.820, Y  +634.626, Z    +0.000, E1   +60.916, E3 +138722.413}
SPL {X  -162.820, Y  +600.578, Z    +0.000, E1   +80.831, E3 +138713.071}
SPL {X  -162.820, Y  +567.495, Z    +0.000, E1   +70.620, E3 +138748.195}
SPL {X  -162.820, Y  +416.506, Z    +0.000, E1   +71.398, E3 +138832.541}
SPL {X  -162.820, Y  +411.010, Z    +0.000, E1   +70.614, E3 +138843.992}
SPL {X  -162.820, Y  +399.588, Z    +0.000, E1   +70.462, E3 +138853.765}
SPL {X  -159.703, Y  +348.793, Z    +0.000, E1   +73.194, E3 +138861.070}
SPL {X  -159.121, Y  +345.992, Z    +0.000, E1   +72.455, E3 +138870.094}
SPL {X  -158.667, Y  +343.959, Z    +0.000, E1   +71.763, E3 +138878.202}
SPL {X  -157.517, Y  +339.284, Z    +0.000, E1   +70.832, E3 +138890.075}
SPL {X  -155.731, Y  +332.978, Z    +0.000, E1   +69.670, E3 +138904.752}
SPL {X  -153.052, Y  +324.954, Z    +0.000, E1   +68.671, E3 +138918.715}
SPL {X  -149.405, Y  +315.782, Z    +0.000, E1   +68.161, E3 +138929.480}
SPL {X  -145.408, Y  +307.240, Z    +0.000, E1   +67.667, E3 +138939.459}
SPL {X  -141.308, Y  +299.614, Z    +0.000, E1   +67.079, E3 +138948.985}
SPL {X  -137.907, Y  +293.943, Z    +0.000, E1   +66.608, E3 +138955.964}
SPL {X  -134.802, Y  +289.183, Z    +0.000, E1   +66.143, E3 +138962.100}
SPL {X  -131.727, Y  +284.801, Z    +0.000, E1   +65.590, E3 +138968.114}
SPL {X  -128.890, Y  +281.012, Z    +0.000, E1   +65.392, E3 +138971.860}
SPL {X  -121.325, Y  +271.915, Z    +0.000, E1   +67.092, E3 +138971.425}
SPL {X   -79.997, Y  +238.687, Z    +0.000, E1   +54.340, E3 +139130.182}
ENDSPLINE

SPLINE
SPL {X  -139.099, Y  +295.872, Z    +0.000, E1   +47.860, E3 +139258.057}
SPL {X  -156.463, Y  +335.448, Z    +0.000, E1   +33.333, E3 +139268.766}
SPL {X  -161.312, Y  +358.394, Z    +0.000, E1   +19.478, E3 +139270.400}
SPL {X  -162.549, Y  +371.111, Z    +0.000, E1    +9.905, E3 +139270.460}
SPL {X  -162.818, Y  +379.769, Z    +0.000, E1    +2.607, E3 +139270.202}
SPL {X  -162.820, Y  +382.500, Z    +0.000, E1    +0.000, E3 +139269.772}
SPL {X  -162.820, Y  +383.721, Z    +0.000, E1    -1.897, E3 +139269.509}
SPL {X  -162.820, Y  +387.689, Z    +0.000, E1    -9.147, E3 +139269.405}
SPL {X  -162.820, Y  +392.805, Z    +0.000, E1   -19.930, E3 +139269.379}
SPL {X  -162.820, Y  +397.742, Z    +0.000, E1   -30.068, E3 +139269.411}
SPL {X  -162.820, Y  +403.938, Z    +0.000, E1   -41.112, E3 +139269.390}
SPL {X  -162.820, Y  +415.430, Z    +0.000, E1   -55.307, E3 +139269.590}
SPL {X  -162.820, Y  +466.986, Z    +0.000, E1   -71.397, E3 +139281.349}
SPL {X  -162.820, Y  +661.594, Z    +0.000, E1   -73.988, E3 +139366.975}
ENDSPLINE

SPLINE
SPL {X  -162.820, Y  +646.360, Z    +0.000, E1   -70.938, E3 +139388.106}
ENDSPLINE

SPLINE
SPL {X  -162.820, Y  +667.477, Z    +0.000, E1   -70.889, E3 +139403.621}
SPL {X  -162.462, Y  +684.286, Z    +0.000, E1   -70.880, E3 +139415.854}
SPL {X  -160.799, Y  +699.074, Z    +0.000, E1   -70.750, E3 +139427.718}
SPL {X  -158.733, Y  +709.754, Z    +0.000, E1   -70.504, E3 +139437.601}
SPL {X  -156.566, Y  +718.194, Z    +0.000, E1   -70.115, E3 +139447.082}
SPL {X  -153.268, Y  +728.449, Z    +0.000, E1   -69.855, E3 +139456.707}
SPL {X  -150.033, Y  +736.750, Z    +0.000, E1   -69.498, E3 +139465.419}
SPL {X  -146.704, Y  +744.128, Z    +0.000, E1   -68.985, E3 +139474.541}
SPL {X  -143.061, Y  +751.243, Z    +0.000, E1   -68.459, E3 +139483.237}
SPL {X  -139.143, Y  +758.055, Z    +0.000, E1   -68.038, E3 +139490.799}
SPL {X  -134.977, Y  +764.558, Z    +0.000, E1   -67.353, E3 +139499.370}
SPL {X  -130.728, Y  +770.560, Z    +0.000, E1   -66.612, E3 +139507.406}
SPL {X  -127.384, Y  +774.909, Z    +0.000, E1   -66.413, E3 +139511.348}
SPL {X  -122.177, Y  +781.125, Z    +0.000, E1   -67.611, E3 +139510.717}
SPL {X   -78.323, Y  +816.244, Z    +0.000, E1   -56.979, E3 +139618.226}
ENDSPLINE

SPLINE
SPL {X   -93.623, Y  +806.710, Z    +0.000, E1   -55.511, E3 +139763.913}
SPL {X  -143.027, Y  +751.304, Z    +0.000, E1   -47.932, E3 +139813.973}
SPL {X  -157.876, Y  +713.320, Z    +0.000, E1   -31.448, E3 +139816.931}
SPL {X  -161.323, Y  +695.531, Z    +0.000, E1   -20.168, E3 +139818.974}
SPL {X  -162.428, Y  +684.786, Z    +0.000, E1   -11.829, E3 +139818.871}
SPL {X  -162.809, Y  +675.372, Z    +0.000, E1    -3.788, E3 +139818.986}
SPL {X  -162.820, Y  +671.476, Z    +0.000, E1    +0.020, E3 +139818.499}
SPL {X  -162.820, Y  +668.959, Z    +0.000, E1    +4.387, E3 +139818.220}
SPL {X  -162.820, Y  +664.344, Z    +0.000, E1   +14.120, E3 +139818.118}
SPL {X  -162.820, Y  +658.993, Z    +0.000, E1   +25.845, E3 +139818.208}
SPL {X  -162.820, Y  +652.443, Z    +0.000, E1   +38.206, E3 +139818.944}
SPL {X  -162.820, Y  +640.832, Z    +0.000, E1   +55.385, E3 +139817.657}
SPL {X  -162.820, Y  +617.334, Z    +0.000, E1   +73.158, E3 +139813.971}
SPL {X  -162.820, Y  +567.495, Z    +0.000, E1   +70.620, E3 +139843.433}
SPL {X  -162.820, Y  +406.037, Z    +0.000, E1   +72.667, E3 +139922.170}
ENDSPLINE

SPLINE
SPL {X  -162.820, Y  +414.365, Z    +0.000, E1   +70.598, E3 +139937.016}
ENDSPLINE

SPLINE
SPL {X  -162.820, Y  +399.588, Z    +0.000, E1   +70.462, E3 +139949.003}
SPL {X  -159.703, Y  +348.793, Z    +0.000, E1   +73.194, E3 +139956.308}
SPL {X  -159.121, Y  +345.992, Z    +0.000, E1   +72.455, E3 +139965.332}
SPL {X  -158.667, Y  +343.959, Z    +0.000, E1   +71.763, E3 +139973.440}
SPL {X  -157.517, Y  +339.284, Z    +0.000, E1   +70.832, E3 +139985.313}
SPL {X  -155.731, Y  +332.978, Z    +0.000, E1   +69.670, E3 +139999.990}
SPL {X  -154.241, Y  +328.346, Z    +0.000, E1   +68.710, E3 +140010.933}
SPL {X  -151.364, Y  +320.507, Z    +0.000, E1   +68.513, E3 +140018.559}
SPL {X  -147.865, Y  +312.336, Z    +0.000, E1   +67.945, E3 +140028.849}
SPL {X  -144.739, Y  +305.928, Z    +0.000, E1   +67.540, E3 +140036.433}
SPL {X  -141.308, Y  +299.614, Z    +0.000, E1   +67.079, E3 +140044.223}
SPL {X  -137.907, Y  +293.943, Z    +0.000, E1   +66.608, E3 +140051.202}
SPL {X  -134.802, Y  +289.183, Z    +0.000, E1   +66.143, E3 +140057.338}
SPL {X  -131.727, Y  +284.801, Z    +0.000, E1   +65.590, E3 +140063.352}
SPL {X  -128.890, Y  +281.012, Z    +0.000, E1   +65.392, E3 +140067.098}
SPL {X  -121.325, Y  +271.915, Z    +0.000, E1   +67.092, E3 +140066.664}
SPL {X   -79.997, Y  +238.687, Z    +0.000, E1   +54.340, E3 +140225.420}
ENDSPLINE

SPLINE
SPL {X  -139.099, Y  +295.872, Z    +0.000, E1   +47.860, E3 +140353.295}
SPL {X  -156.463, Y  +335.448, Z    +0.000, E1   +33.333, E3 +140364.004}
SPL {X  -161.312, Y  +358.394, Z    +0.000, E1   +19.478, E3 +140365.638}
SPL {X  -162.549, Y  +371.111, Z    +0.000, E1    +9.905, E3 +140365.698}
SPL {X  -162.818, Y  +379.769, Z    +0.000, E1    +2.607, E3 +140365.440}
SPL {X  -162.820, Y  +382.897, Z    +0.000, E1    -0.379, E3 +140364.924}
SPL {X  -162.820, Y  +387.689, Z    +0.000, E1    -9.147, E3 +140364.643}
SPL {X  -162.820, Y  +392.805, Z    +0.000, E1   -19.930, E3 +140364.617}
SPL {X  -162.820, Y  +397.742, Z    +0.000, E1   -30.068, E3 +140364.649}
SPL {X  -162.820, Y  +403.938, Z    +0.000, E1   -41.112, E3 +140364.629}
SPL {X  -162.820, Y  +415.430, Z    +0.000, E1   -55.307, E3 +140364.828}
SPL {X  -162.820, Y  +466.986, Z    +0.000, E1   -71.397, E3 +140376.587}
SPL {X  -162.820, Y  +661.594, Z    +0.000, E1   -73.988, E3 +140462.213}
ENDSPLINE

SPLINE
SPL {X  -162.820, Y  +634.363, Z    +0.000, E1   -70.793, E3 +140475.791}
ENDSPLINE

SPLINE
SPL {X  -162.820, Y  +649.777, Z    +0.000, E1   -70.953, E3 +140485.550}
SPL {X  -162.820, Y  +667.477, Z    +0.000, E1   -70.889, E3 +140498.859}
SPL {X  -162.097, Y  +688.831, Z    +0.000, E1   -70.910, E3 +140514.230}
SPL {X  -159.319, Y  +707.081, Z    +0.000, E1   -70.563, E3 +140530.516}
SPL {X  -156.566, Y  +718.194, Z    +0.000, E1   -70.115, E3 +140542.320}
SPL {X  -153.268, Y  +728.449, Z    +0.000, E1   -69.855, E3 +140551.946}
SPL {X  -150.033, Y  +736.750, Z    +0.000, E1   -69.498, E3 +140560.657}
SPL {X  -146.704, Y  +744.128, Z    +0.000, E1   -68.985, E3 +140569.779}
SPL {X  -142.102, Y  +752.982, Z    +0.000, E1   -68.357, E3 +140580.518}
SPL {X  -138.073, Y  +759.791, Z    +0.000, E1   -67.958, E3 +140587.687}
SPL {X  -134.977, Y  +764.558, Z    +0.000, E1   -67.353, E3 +140594.609}
SPL {X  -130.728, Y  +770.560, Z    +0.000, E1   -66.612, E3 +140602.644}
SPL {X  -125.283, Y  +777.493, Z    +0.000, E1   -66.879, E3 +140606.369}
SPL {X   -78.323, Y  +816.244, Z    +0.000, E1   -56.979, E3 +140713.465}
ENDSPLINE

SPLINE
SPL {X   -93.623, Y  +806.710, Z    +0.000, E1   -55.511, E3 +140859.151}
SPL {X  -143.027, Y  +751.304, Z    +0.000, E1   -47.932, E3 +140909.211}
SPL {X  -157.876, Y  +713.320, Z    +0.000, E1   -31.448, E3 +140912.169}
SPL {X  -161.323, Y  +695.531, Z    +0.000, E1   -20.168, E3 +140914.212}
SPL {X  -162.626, Y  +681.447, Z    +0.000, E1    -9.120, E3 +140914.201}
SPL {X  -162.820, Y  +671.283, Z    +0.000, E1    +0.049, E3 +140913.713}
SPL {X  -162.820, Y  +665.565, Z    +0.000, E1   +11.206, E3 +140913.376}
SPL {X  -162.820, Y  +658.993, Z    +0.000, E1   +25.845, E3 +140913.446}
SPL {X  -162.820, Y  +650.479, Z    +0.000, E1   +41.861, E3 +140913.606}
SPL {X  -162.820, Y  +634.626, Z    +0.000, E1   +60.916, E3 +140912.889}
SPL {X  -162.820, Y  +600.578, Z    +0.000, E1   +80.831, E3 +140903.547}
SPL {X  -162.820, Y  +567.495, Z    +0.000, E1   +70.620, E3 +140938.671}
SPL {X  -162.820, Y  +416.506, Z    +0.000, E1   +71.398, E3 +141023.017}
SPL {X  -162.820, Y  +411.010, Z    +0.000, E1   +70.614, E3 +141034.468}
SPL {X  -162.820, Y  +399.588, Z    +0.000, E1   +70.462, E3 +141044.242}
SPL {X  -159.703, Y  +348.793, Z    +0.000, E1   +73.194, E3 +141051.546}
SPL {X  -159.121, Y  +345.992, Z    +0.000, E1   +72.455, E3 +141060.570}
SPL {X  -158.667, Y  +343.959, Z    +0.000, E1   +71.763, E3 +141068.678}
SPL {X  -157.517, Y  +339.284, Z    +0.000, E1   +70.832, E3 +141080.551}
SPL {X  -155.731, Y  +332.978, Z    +0.000, E1   +69.670, E3 +141095.228}
SPL {X  -153.052, Y  +324.954, Z    +0.000, E1   +68.671, E3 +141109.191}
SPL {X  -149.405, Y  +315.782, Z    +0.000, E1   +68.161, E3 +141119.956}
SPL {X  -145.408, Y  +307.240, Z    +0.000, E1   +67.667, E3 +141129.935}
SPL {X  -141.308, Y  +299.614, Z    +0.000, E1   +67.079, E3 +141139.462}
SPL {X  -137.907, Y  +293.943, Z    +0.000, E1   +66.608, E3 +141146.440}
SPL {X  -134.802, Y  +289.183, Z    +0.000, E1   +66.143, E3 +141152.576}
SPL {X  -131.727, Y  +284.801, Z    +0.000, E1   +65.590, E3 +141158.591}
SPL {X  -128.890, Y  +281.012, Z    +0.000, E1   +65.392, E3 +141162.336}
SPL {X  -121.325, Y  +271.915, Z    +0.000, E1   +67.092, E3 +141161.902}
SPL {X   -79.997, Y  +238.687, Z    +0.000, E1   +54.340, E3 +141320.658}
ENDSPLINE

SPLINE
SPL {X  -139.099, Y  +295.872, Z    +0.000, E1   +47.860, E3 +141448.534}
SPL {X  -156.463, Y  +335.448, Z    +0.000, E1   +33.333, E3 +141459.242}
SPL {X  -161.312, Y  +358.394, Z    +0.000, E1   +19.478, E3 +141460.876}
SPL {X  -162.549, Y  +371.111, Z    +0.000, E1    +9.905, E3 +141460.936}
SPL {X  -162.818, Y  +379.769, Z    +0.000, E1    +2.607, E3 +141460.678}
SPL {X  -162.820, Y  +382.897, Z    +0.000, E1    -0.379, E3 +141460.162}
SPL {X  -162.820, Y  +387.689, Z    +0.000, E1    -9.147, E3 +141459.882}
SPL {X  -162.820, Y  +392.805, Z    +0.000, E1   -19.930, E3 +141459.855}
SPL {X  -162.820, Y  +397.742, Z    +0.000, E1   -30.068, E3 +141459.887}
SPL {X  -162.820, Y  +403.938, Z    +0.000, E1   -41.112, E3 +141459.867}
SPL {X  -162.820, Y  +415.430, Z    +0.000, E1   -55.307, E3 +141460.066}
SPL {X  -162.820, Y  +466.986, Z    +0.000, E1   -71.397, E3 +141471.825}
SPL {X  -162.820, Y  +661.594, Z    +0.000, E1   -73.988, E3 +141557.451}
ENDSPLINE

SPLINE
SPL {X  -162.820, Y  +634.363, Z    +0.000, E1   -70.793, E3 +141571.029}
ENDSPLINE

SPLINE
SPL {X  -162.820, Y  +649.777, Z    +0.000, E1   -70.953, E3 +141580.788}
SPL {X  -162.820, Y  +667.477, Z    +0.000, E1   -70.889, E3 +141594.097}
SPL {X  -162.462, Y  +684.286, Z    +0.000, E1   -70.880, E3 +141606.330}
SPL {X  -160.799, Y  +699.074, Z    +0.000, E1   -70.750, E3 +141618.194}
SPL {X  -158.733, Y  +709.754, Z    +0.000, E1   -70.504, E3 +141628.077}
SPL {X  -156.566, Y  +718.194, Z    +0.000, E1   -70.115, E3 +141637.558}
SPL {X  -153.268, Y  +728.449, Z    +0.000, E1   -69.855, E3 +141647.184}
SPL {X  -150.033, Y  +736.750, Z    +0.000, E1   -69.498, E3 +141655.895}
SPL {X  -146.704, Y  +744.128, Z    +0.000, E1   -68.985, E3 +141665.017}
SPL {X  -143.061, Y  +751.243, Z    +0.000, E1   -68.459, E3 +141673.713}
SPL {X  -139.143, Y  +758.055, Z    +0.000, E1   -68.038, E3 +141681.276}
SPL {X  -134.977, Y  +764.558, Z    +0.000, E1   -67.353, E3 +141689.847}
SPL {X  -130.728, Y  +770.560, Z    +0.000, E1   -66.612, E3 +141697.882}
SPL {X  -125.283, Y  +777.493, Z    +0.000, E1   -66.879, E3 +141701.607}
SPL {X   -78.323, Y  +816.244, Z    +0.000, E1   -56.979, E3 +141808.703}
ENDSPLINE

SPLINE
SPL {X   -93.623, Y  +806.710, Z    +0.000, E1   -55.511, E3 +141954.389}
SPL {X  -138.493, Y  +759.115, Z    +0.000, E1   -50.023, E3 +142002.217}
SPL {X  -149.871, Y  +737.133, Z    +0.000, E1   -43.112, E3 +142007.631}
SPL {X  -157.876, Y  +713.320, Z    +0.000, E1   -31.448, E3 +142007.407}
SPL {X  -161.323, Y  +695.531, Z    +0.000, E1   -20.168, E3 +142009.450}
SPL {X  -162.428, Y  +684.786, Z    +0.000, E1   -11.829, E3 +142009.347}
SPL {X  -162.809, Y  +675.372, Z    +0.000, E1    -3.788, E3 +142009.462}
SPL {X  -162.820, Y  +671.476, Z    +0.000, E1    +0.020, E3 +142008.975}
SPL {X  -162.820, Y  +668.959, Z    +0.000, E1    +4.387, E3 +142008.696}
SPL {X  -162.820, Y  +664.344, Z    +0.000, E1   +14.120, E3 +142008.595}
SPL {X  -162.820, Y  +658.993, Z    +0.000, E1   +25.845, E3 +142008.685}
SPL {X  -162.820, Y  +650.479, Z    +0.000, E1   +41.861, E3 +142008.844}
SPL {X  -162.820, Y  +634.626, Z    +0.000, E1   +60.916, E3 +142008.127}
SPL {X  -162.820, Y  +600.578, Z    +0.000, E1   +80.831, E3 +141998.785}
SPL {X  -162.820, Y  +567.495, Z    +0.000, E1   +70.620, E3 +142033.909}
SPL {X  -162.820, Y  +416.506, Z    +0.000, E1   +71.398, E3 +142118.255}
SPL {X  -162.820, Y  +411.010, Z    +0.000, E1   +70.614, E3 +142129.706}
SPL {X  -162.820, Y  +399.588, Z    +0.000, E1   +70.462, E3 +142139.480}
SPL {X  -159.703, Y  +348.793, Z    +0.000, E1   +73.194, E3 +142146.784}
SPL {X  -158.911, Y  +345.038, Z    +0.000, E1   +72.209, E3 +142159.000}
SPL {X  -158.117, Y  +341.649, Z    +0.000, E1   +71.181, E3 +142170.957}
SPL {X  -156.755, Y  +336.473, Z    +0.000, E1   +70.264, E3 +142182.732}
SPL {X  -155.322, Y  +331.660, Z    +0.000, E1   +69.461, E3 +142192.979}
SPL {X  -153.052, Y  +324.954, Z    +0.000, E1   +68.671, E3 +142204.429}
SPL {X  -149.405, Y  +315.782, Z    +0.000, E1   +68.161, E3 +142215.194}
SPL {X  -145.408, Y  +307.240, Z    +0.000, E1   +67.667, E3 +142225.173}
SPL {X  -141.308, Y  +299.614, Z    +0.000, E1   +67.079, E3 +142234.700}
SPL {X  -137.907, Y  +293.943, Z    +0.000, E1   +66.608, E3 +142241.678}
SPL {X  -134.802, Y  +289.183, Z    +0.000, E1   +66.143, E3 +142247.814}
SPL {X  -131.727, Y  +284.801, Z    +0.000, E1   +65.590, E3 +142253.829}
SPL {X  -128.890, Y  +281.012, Z    +0.000, E1   +65.392, E3 +142257.574}
SPL {X  -121.325, Y  +271.915, Z    +0.000, E1   +67.092, E3 +142257.140}
SPL {X   -79.997, Y  +238.687, Z    +0.000, E1   +54.340, E3 +142415.896}
ENDSPLINE

SPLINE
SPL {X  -139.099, Y  +295.872, Z    +0.000, E1   +47.860, E3 +142543.772}
SPL {X  -156.463, Y  +335.448, Z    +0.000, E1   +33.333, E3 +142554.480}
SPL {X  -161.312, Y  +358.394, Z    +0.000, E1   +19.478, E3 +142556.115}
SPL {X  -162.549, Y  +371.111, Z    +0.000, E1    +9.905, E3 +142556.174}
SPL {X  -162.818, Y  +379.769, Z    +0.000, E1    +2.607, E3 +142555.916}
SPL {X  -162.820, Y  +382.500, Z    +0.000, E1    +0.000, E3 +142555.486}
SPL {X  -162.820, Y  +383.721, Z    +0.000, E1    -1.897, E3 +142555.223}
SPL {X  -162.820, Y  +387.689, Z    +0.000, E1    -9.147, E3 +142555.120}
SPL {X  -162.820, Y  +392.805, Z    +0.000, E1   -19.930, E3 +142555.093}
SPL {X  -162.820, Y  +397.742, Z    +0.000, E1   -30.068, E3 +142555.125}
SPL {X  -162.820, Y  +403.938, Z    +0.000, E1   -41.112, E3 +142555.105}
SPL {X  -162.820, Y  +415.430, Z    +0.000, E1   -55.307, E3 +142555.304}
SPL {X  -162.820, Y  +466.986, Z    +0.000, E1   -71.397, E3 +142567.063}
SPL {X  -162.820, Y  +661.594, Z    +0.000, E1   -73.988, E3 +142652.689}
ENDSPLINE

SPLINE
SPL {X  -162.820, Y  +646.360, Z    +0.000, E1   -70.938, E3 +142673.820}
ENDSPLINE

SPLINE
SPL {X  -162.820, Y  +667.477, Z    +0.000, E1   -70.889, E3 +142689.335}
SPL {X  -162.462, Y  +684.286, Z    +0.000, E1   -70.880, E3 +142701.568}
SPL {X  -160.799, Y  +699.074, Z    +0.000, E1   -70.750, E3 +142713.432}
SPL {X  -158.733, Y  +709.754, Z    +0.000, E1   -70.504, E3 +142723.315}
SPL {X  -155.769, Y  +720.894, Z    +0.000, E1   -70.077, E3 +142735.202}
SPL {X  -152.498, Y  +730.550, Z    +0.000, E1   -69.764, E3 +142744.568}
SPL {X  -149.282, Y  +738.502, Z    +0.000, E1   -69.318, E3 +142753.943}
SPL {X  -145.460, Y  +746.655, Z    +0.000, E1   -68.995, E3 +142761.957}
SPL {X  -142.102, Y  +752.982, Z    +0.000, E1   -68.357, E3 +142770.994}
SPL {X  -138.073, Y  +759.791, Z    +0.000, E1   -67.958, E3 +142778.164}
SPL {X  -134.977, Y  +764.558, Z    +0.000, E1   -67.353, E3 +142785.085}
SPL {X  -130.728, Y  +770.560, Z    +0.000, E1   -66.612, E3 +142793.120}
SPL {X  -125.283, Y  +777.493, Z    +0.000, E1   -66.879, E3 +142796.845}
SPL {X   -78.323, Y  +816.244, Z    +0.000, E1   -56.979, E3 +142903.941}
ENDSPLINE

SPLINE
SPL {X   -93.623, Y  +806.710, Z    +0.000, E1   -55.511, E3 +143049.627}
SPL {X  -138.493, Y  +759.115, Z    +0.000, E1   -50.023, E3 +143097.455}
SPL {X  -149.871, Y  +737.133, Z    +0.000, E1   -43.112, E3 +143102.869}
SPL {X  -157.876, Y  +713.320, Z    +0.000, E1   -31.448, E3 +143102.645}
SPL {X  -161.323, Y  +695.531, Z    +0.000, E1   -20.168, E3 +143104.688}
SPL {X  -162.626, Y  +681.447, Z    +0.000, E1    -9.120, E3 +143104.677}
SPL {X  -162.820, Y  +673.597, Z    +0.000, E1    -2.055, E3 +143104.671}
SPL {X  -162.820, Y  +671.476, Z    +0.000, E1    +0.020, E3 +143104.213}
SPL {X  -162.820, Y  +668.959, Z    +0.000, E1    +4.387, E3 +143103.934}
SPL {X  -162.820, Y  +664.344, Z    +0.000, E1   +14.120, E3 +143103.833}
SPL {X  -162.820, Y  +658.993, Z    +0.000, E1   +25.845, E3 +143103.923}
SPL {X  -162.820, Y  +652.443, Z    +0.000, E1   +38.206, E3 +143104.658}
SPL {X  -162.820, Y  +640.832, Z    +0.000, E1   +55.385, E3 +143103.372}
SPL {X  -162.820, Y  +617.334, Z    +0.000, E1   +73.158, E3 +143099.686}
SPL {X  -162.820, Y  +567.495, Z    +0.000, E1   +70.620, E3 +143129.147}
SPL {X  -162.820, Y  +416.506, Z    +0.000, E1   +71.398, E3 +143213.493}
SPL {X  -162.820, Y  +411.010, Z    +0.000, E1   +70.614, E3 +143224.944}
SPL {X  -162.820, Y  +391.151, Z    +0.000, E1   +70.927, E3 +143236.399}
SPL {X  -159.025, Y  +345.550, Z    +0.000, E1   +73.389, E3 +143242.080}
SPL {X  -158.911, Y  +345.038, Z    +0.000, E1   +72.209, E3 +143254.238}
SPL {X  -157.738, Y  +340.137, Z    +0.000, E1   +71.006, E3 +143269.055}
SPL {X  -155.731, Y  +332.978, Z    +0.000, E1   +69.670, E3 +143285.705}
SPL {X  -153.052, Y  +324.954, Z    +0.000, E1   +68.671, E3 +143299.667}
SPL {X  -148.581, Y  +313.911, Z    +0.000, E1   +68.095, E3 +143312.457}
SPL {X  -143.686, Y  +303.920, Z    +0.000, E1   +67.419, E3 +143324.594}
SPL {X  -138.888, Y  +295.526, Z    +0.000, E1   +66.767, E3 +143334.928}
SPL {X  -134.802, Y  +289.183, Z    +0.000, E1   +66.143, E3 +143343.052}
SPL {X  -131.727, Y  +284.801, Z    +0.000, E1   +65.590, E3 +143349.067}
SPL {X  -128.890, Y  +281.012, Z    +0.000, E1   +65.392, E3 +143352.812}
SPL {X  -121.325, Y  +271.915, Z    +0.000, E1   +67.092, E3 +143352.378}
SPL {X   -79.997, Y  +238.687, Z    +0.000, E1   +54.340, E3 +143511.134}
ENDSPLINE

SPLINE
SPL {X  -139.099, Y  +295.872, Z    +0.000, E1   +47.860, E3 +143639.010}
SPL {X  -156.463, Y  +335.448, Z    +0.000, E1   +33.333, E3 +143649.718}
SPL {X  -161.312, Y  +358.394, Z    +0.000, E1   +19.478, E3 +143651.353}
SPL {X  -162.549, Y  +371.111, Z    +0.000, E1    +9.905, E3 +143651.412}
SPL {X  -162.818, Y  +379.769, Z    +0.000, E1    +2.607, E3 +143651.154}
SPL {X  -162.820, Y  +382.500, Z    +0.000, E1    +0.000, E3 +143650.724}
SPL {X  -162.820, Y  +384.989, Z    +0.000, E1    -3.865, E3 +143650.451}
SPL {X  -162.820, Y  +391.404, Z    +0.000, E1   -16.767, E3 +143650.298}
SPL {X  -162.820, Y  +397.742, Z    +0.000, E1   -30.068, E3 +143650.363}
SPL {X  -162.820, Y  +403.938, Z    +0.000, E1   -41.112, E3 +143650.343}
SPL {X  -162.820, Y  +415.430, Z    +0.000, E1   -55.307, E3 +143650.542}
SPL {X  -162.820, Y  +466.986, Z    +0.000, E1   -71.397, E3 +143662.301}
SPL {X  -162.820, Y  +661.594, Z    +0.000, E1   -73.988, E3 +143747.928}
ENDSPLINE

SPLINE
SPL {X  -162.820, Y  +639.523, Z    +0.000, E1   -70.828, E3 +143765.004}
ENDSPLINE

SPLINE
SPL {X  -162.820, Y  +655.227, Z    +0.000, E1   -71.020, E3 +143774.430}
SPL {X  -162.820, Y  +667.477, Z    +0.000, E1   -70.889, E3 +143784.573}
SPL {X  -162.097, Y  +688.831, Z    +0.000, E1   -70.910, E3 +143799.944}
SPL {X  -159.319, Y  +707.081, Z    +0.000, E1   -70.563, E3 +143816.230}
SPL {X  -155.769, Y  +720.894, Z    +0.000, E1   -70.077, E3 +143830.440}
SPL {X  -150.995, Y  +734.417, Z    +0.000, E1   -69.635, E3 +143843.816}
SPL {X  -146.704, Y  +744.128, Z    +0.000, E1   -68.985, E3 +143855.494}
SPL {X  -142.102, Y  +752.982, Z    +0.000, E1   -68.357, E3 +143866.232}
SPL {X  -138.073, Y  +759.791, Z    +0.000, E1   -67.958, E3 +143873.402}
SPL {X  -134.977, Y  +764.558, Z    +0.000, E1   -67.353, E3 +143880.323}
SPL {X  -130.728, Y  +770.560, Z    +0.000, E1   -66.612, E3 +143888.358}
SPL {X  -125.283, Y  +777.493, Z    +0.000, E1   -66.879, E3 +143892.083}
SPL {X   -78.323, Y  +816.244, Z    +0.000, E1   -56.979, E3 +143999.179}
ENDSPLINE

SPLINE
SPL {X   -93.623, Y  +806.710, Z    +0.000, E1   -55.511, E3 +144144.865}
SPL {X  -143.027, Y  +751.304, Z    +0.000, E1   -47.932, E3 +144194.926}
SPL {X  -157.876, Y  +713.320, Z    +0.000, E1   -31.448, E3 +144197.883}
SPL {X  -161.323, Y  +695.531, Z    +0.000, E1   -20.168, E3 +144199.927}
SPL {X  -162.626, Y  +681.447, Z    +0.000, E1    -9.120, E3 +144199.915}
SPL {X  -162.820, Y  +673.597, Z    +0.000, E1    -2.055, E3 +144199.909}
SPL {X  -162.820, Y  +671.122, Z    +0.000, E1    +0.366, E3 +144199.394}
SPL {X  -162.820, Y  +665.565, Z    +0.000, E1   +11.206, E3 +144199.091}
SPL {X  -162.820, Y  +658.993, Z    +0.000, E1   +25.845, E3 +144199.161}
SPL {X  -162.820, Y  +650.479, Z    +0.000, E1   +41.861, E3 +144199.320}
SPL {X  -162.820, Y  +634.626, Z    +0.000, E1   +60.916, E3 +144198.603}
SPL {X  -162.820, Y  +600.578, Z    +0.000, E1   +80.831, E3 +144189.261}
SPL {X  -162.820, Y  +567.495, Z    +0.000, E1   +70.620, E3 +144224.386}
SPL {X  -162.820, Y  +416.506, Z    +0.000, E1   +71.398, E3 +144308.731}
SPL {X  -162.820, Y  +411.010, Z    +0.000, E1   +70.614, E3 +144320.182}
SPL {X  -162.820, Y  +399.588, Z    +0.000, E1   +70.462, E3 +144329.956}
SPL {X  -159.703, Y  +348.793, Z    +0.000, E1   +73.194, E3 +144337.260}
SPL {X  -158.809, Y  +344.584, Z    +0.000, E1   +72.042, E3 +144351.565}
SPL {X  -157.517, Y  +339.284, Z    +0.000, E1   +70.832, E3 +144366.266}
SPL {X  -155.731, Y  +332.978, Z    +0.000, E1   +69.670, E3 +144380.943}
SPL {X  -153.052, Y  +324.954, Z    +0.000, E1   +68.671, E3 +144394.905}
SPL {X  -149.405, Y  +315.782, Z    +0.000, E1   +68.161, E3 +144405.671}
SPL {X  -145.408, Y  +307.240, Z    +0.000, E1   +67.667, E3 +144415.649}
SPL {X  -141.308, Y  +299.614, Z    +0.000, E1   +67.079, E3 +144425.176}
SPL {X  -137.907, Y  +293.943, Z    +0.000, E1   +66.608, E3 +144432.154}
SPL {X  -134.802, Y  +289.183, Z    +0.000, E1   +66.143, E3 +144438.290}
SPL {X  -131.727, Y  +284.801, Z    +0.000, E1   +65.590, E3 +144444.305}
SPL {X  -128.890, Y  +281.012, Z    +0.000, E1   +65.392, E3 +144448.050}
SPL {X  -121.325, Y  +271.915, Z    +0.000, E1   +67.092, E3 +144447.616}
SPL {X   -79.997, Y  +238.687, Z    +0.000, E1   +54.340, E3 +144606.372}
ENDSPLINE

SPLINE
SPL {X  -139.099, Y  +295.872, Z    +0.000, E1   +47.860, E3 +144734.248}
SPL {X  -156.463, Y  +335.448, Z    +0.000, E1   +33.333, E3 +144744.956}
SPL {X  -161.312, Y  +358.394, Z    +0.000, E1   +19.478, E3 +144746.591}
SPL {X  -162.549, Y  +371.111, Z    +0.000, E1    +9.905, E3 +144746.650}
SPL {X  -162.818, Y  +379.769, Z    +0.000, E1    +2.607, E3 +144746.393}
SPL {X  -162.820, Y  +382.500, Z    +0.000, E1    +0.000, E3 +144745.962}
SPL {X  -162.820, Y  +383.721, Z    +0.000, E1    -1.897, E3 +144745.699}
SPL {X  -162.820, Y  +387.689, Z    +0.000, E1    -9.147, E3 +144745.596}
SPL {X  -162.820, Y  +392.805, Z    +0.000, E1   -19.930, E3 +144745.569}
SPL {X  -162.820, Y  +397.742, Z    +0.000, E1   -30.068, E3 +144745.601}
SPL {X  -162.820, Y  +403.938, Z    +0.000, E1   -41.112, E3 +144745.581}
SPL {X  -162.820, Y  +415.430, Z    +0.000, E1   -55.307, E3 +144745.780}
SPL {X  -162.820, Y  +466.986, Z    +0.000, E1   -71.397, E3 +144757.539}
SPL {X  -162.820, Y  +661.594, Z    +0.000, E1   -73.988, E3 +144843.166}
ENDSPLINE

SPLINE
SPL {X  -162.820, Y  +646.360, Z    +0.000, E1   -70.938, E3 +144864.296}
ENDSPLINE

SPLINE
SPL {X  -162.820, Y  +667.477, Z    +0.000, E1   -70.889, E3 +144879.811}
SPL {X  -162.462, Y  +684.286, Z    +0.000, E1   -70.880, E3 +144892.044}
SPL {X  -160.799, Y  +699.074, Z    +0.000, E1   -70.750, E3 +144903.908}
SPL {X  -158.733, Y  +709.754, Z    +0.000, E1   -70.504, E3 +144913.791}
SPL {X  -155.769, Y  +720.894, Z    +0.000, E1   -70.077, E3 +144925.678}
SPL {X  -152.498, Y  +730.550, Z    +0.000, E1   -69.764, E3 +144935.044}
SPL {X  -149.282, Y  +738.502, Z    +0.000, E1   -69.318, E3 +144944.419}
SPL {X  -145.460, Y  +746.655, Z    +0.000, E1   -68.995, E3 +144952.433}
SPL {X  -142.102, Y  +752.982, Z    +0.000, E1   -68.357, E3 +144961.470}
SPL {X  -136.987, Y  +761.506, Z    +0.000, E1   -67.725, E3 +144971.355}
SPL {X  -133.055, Y  +767.344, Z    +0.000, E1   -67.024, E3 +144979.256}
SPL {X  -129.955, Y  +771.593, Z    +0.000, E1   -66.476, E3 +144984.897}
SPL {X  -125.283, Y  +777.493, Z    +0.000, E1   -66.879, E3 +144987.321}
SPL {X   -78.323, Y  +816.244, Z    +0.000, E1   -56.979, E3 +145094.417}
ENDSPLINE

SPLINE
SPL {X   -93.623, Y  +806.710, Z    +0.000, E1   -55.511, E3 +145240.103}
SPL {X  -138.493, Y  +759.115, Z    +0.000, E1   -50.023, E3 +145287.931}
SPL {X  -149.871, Y  +737.133, Z    +0.000, E1   -43.112, E3 +145293.346}
SPL {X  -157.876, Y  +713.320, Z    +0.000, E1   -31.448, E3 +145293.121}
SPL {X  -161.323, Y  +695.531, Z    +0.000, E1   -20.168, E3 +145295.165}
SPL {X  -162.428, Y  +684.786, Z    +0.000, E1   -11.829, E3 +145295.062}
SPL {X  -162.809, Y  +675.372, Z    +0.000, E1    -3.788, E3 +145295.176}
SPL {X  -162.820, Y  +671.476, Z    +0.000, E1    +0.020, E3 +145294.689}
SPL {X  -162.820, Y  +668.959, Z    +0.000, E1    +4.387, E3 +145294.410}
SPL {X  -162.820, Y  +664.344, Z    +0.000, E1   +14.120, E3 +145294.309}
SPL {X  -162.820, Y  +658.993, Z    +0.000, E1   +25.845, E3 +145294.399}
SPL {X  -162.820, Y  +650.479, Z    +0.000, E1   +41.861, E3 +145294.558}
SPL {X  -162.820, Y  +634.626, Z    +0.000, E1   +60.916, E3 +145293.842}
SPL {X  -162.820, Y  +600.578, Z    +0.000, E1   +80.831, E3 +145284.499}
SPL {X  -162.820, Y  +567.495, Z    +0.000, E1   +70.620, E3 +145319.624}
SPL {X  -162.820, Y  +416.506, Z    +0.000, E1   +71.398, E3 +145403.969}
SPL {X  -162.820, Y  +411.010, Z    +0.000, E1   +70.614, E3 +145415.420}
SPL {X  -162.820, Y  +399.588, Z    +0.000, E1   +70.462, E3 +145425.194}
SPL {X  -159.703, Y  +348.793, Z    +0.000, E1   +73.194, E3 +145432.498}
SPL {X  -158.911, Y  +345.038, Z    +0.000, E1   +72.209, E3 +145444.715}
SPL {X  -158.117, Y  +341.649, Z    +0.000, E1   +71.181, E3 +145456.671}
SPL {X  -156.755, Y  +336.473, Z    +0.000, E1   +70.264, E3 +145468.446}
SPL {X  -155.322, Y  +331.660, Z    +0.000, E1   +69.461, E3 +145478.693}
SPL {X  -153.052, Y  +324.954, Z    +0.000, E1   +68.671, E3 +145490.143}
SPL {X  -149.405, Y  +315.782, Z    +0.000, E1   +68.161, E3 +145500.909}
SPL {X  -145.408, Y  +307.240, Z    +0.000, E1   +67.667, E3 +145510.887}
SPL {X  -142.385, Y  +301.526, Z    +0.000, E1   +67.199, E3 +145518.119}
SPL {X  -138.888, Y  +295.526, Z    +0.000, E1   +66.767, E3 +145525.404}
SPL {X  -134.802, Y  +289.183, Z    +0.000, E1   +66.143, E3 +145533.529}
SPL {X  -131.727, Y  +284.801, Z    +0.000, E1   +65.590, E3 +145539.543}
SPL {X  -128.890, Y  +281.012, Z    +0.000, E1   +65.392, E3 +145543.288}
SPL {X  -121.325, Y  +271.915, Z    +0.000, E1   +67.092, E3 +145542.854}
SPL {X   -79.997, Y  +238.687, Z    +0.000, E1   +54.340, E3 +145701.610}
ENDSPLINE

SPLINE
SPL {X  -139.099, Y  +295.872, Z    +0.000, E1   +47.860, E3 +145829.486}
SPL {X  -156.463, Y  +335.448, Z    +0.000, E1   +33.333, E3 +145840.194}
SPL {X  -161.312, Y  +358.394, Z    +0.000, E1   +19.478, E3 +145841.829}
SPL {X  -162.549, Y  +371.111, Z    +0.000, E1    +9.905, E3 +145841.889}
SPL {X  -162.818, Y  +379.769, Z    +0.000, E1    +2.607, E3 +145841.631}
SPL {X  -162.820, Y  +382.897, Z    +0.000, E1    -0.379, E3 +145841.115}
SPL {X  -162.820, Y  +387.689, Z    +0.000, E1    -9.147, E3 +145840.834}
SPL {X  -162.820, Y  +392.805, Z    +0.000, E1   -19.930, E3 +145840.807}
SPL {X  -162.820, Y  +397.742, Z    +0.000, E1   -30.068, E3 +145840.840}
SPL {X  -162.820, Y  +403.938, Z    +0.000, E1   -41.112, E3 +145840.819}
SPL {X  -162.820, Y  +415.430, Z    +0.000, E1   -55.307, E3 +145841.018}
SPL {X  -162.820, Y  +466.986, Z    +0.000, E1   -71.397, E3 +145852.778}
SPL {X  -162.820, Y  +661.594, Z    +0.000, E1   -73.988, E3 +145938.404}
ENDSPLINE

SPLINE
SPL {X  -162.820, Y  +646.360, Z    +0.000, E1   -70.938, E3 +145959.534}
ENDSPLINE

SPLINE
SPL {X  -162.820, Y  +667.477, Z    +0.000, E1   -70.889, E3 +145975.049}
SPL {X  -162.097, Y  +688.831, Z    +0.000, E1   -70.910, E3 +145990.420}
SPL {X  -159.319, Y  +707.081, Z    +0.000, E1   -70.563, E3 +146006.706}
SPL {X  -155.769, Y  +720.894, Z    +0.000, E1   -70.077, E3 +146020.916}
SPL {X  -150.995, Y  +734.417, Z    +0.000, E1   -69.635, E3 +146034.293}
SPL {X  -146.704, Y  +744.128, Z    +0.000, E1   -68.985, E3 +146045.970}
SPL {X  -142.102, Y  +752.982, Z    +0.000, E1   -68.357, E3 +146056.708}
SPL {X  -138.073, Y  +759.791, Z    +0.000, E1   -67.958, E3 +146063.878}
SPL {X  -134.977, Y  +764.558, Z    +0.000, E1   -67.353, E3 +146070.799}
SPL {X  -130.728, Y  +770.560, Z    +0.000, E1   -66.612, E3 +146078.834}
SPL {X  -127.384, Y  +774.909, Z    +0.000, E1   -66.413, E3 +146082.777}
SPL {X  -122.177, Y  +781.125, Z    +0.000, E1   -67.611, E3 +146082.146}
SPL {X   -78.323, Y  +816.244, Z    +0.000, E1   -56.979, E3 +146189.655}
ENDSPLINE

SPLINE
SPL {X   -93.623, Y  +806.710, Z    +0.000, E1   -55.511, E3 +146335.341}
SPL {X  -143.027, Y  +751.304, Z    +0.000, E1   -47.932, E3 +146385.402}
SPL {X  -157.876, Y  +713.320, Z    +0.000, E1   -31.448, E3 +146388.359}
SPL {X  -161.323, Y  +695.531, Z    +0.000, E1   -20.168, E3 +146390.403}
SPL {X  -162.428, Y  +684.786, Z    +0.000, E1   -11.829, E3 +146390.300}
SPL {X  -162.809, Y  +675.372, Z    +0.000, E1    -3.788, E3 +146390.414}
SPL {X  -162.820, Y  +671.476, Z    +0.000, E1    +0.020, E3 +146389.927}
SPL {X  -162.820, Y  +668.959, Z    +0.000, E1    +4.387, E3 +146389.648}
SPL {X  -162.820, Y  +664.344, Z    +0.000, E1   +14.120, E3 +146389.547}
SPL {X  -162.820, Y  +658.993, Z    +0.000, E1   +25.845, E3 +146389.637}
SPL {X  -162.820, Y  +652.443, Z    +0.000, E1   +38.206, E3 +146390.373}
SPL {X  -162.820, Y  +640.832, Z    +0.000, E1   +55.385, E3 +146389.086}
SPL {X  -162.820, Y  +625.562, Z    +0.000, E1   +67.658, E3 +146388.139}
SPL {X  -162.820, Y  +600.578, Z    +0.000, E1   +80.831, E3 +146379.737}
SPL {X  -162.820, Y  +567.495, Z    +0.000, E1   +70.620, E3 +146414.862}
SPL {X  -162.820, Y  +416.506, Z    +0.000, E1   +71.398, E3 +146499.207}
SPL {X  -162.820, Y  +411.010, Z    +0.000, E1   +70.614, E3 +146510.659}
SPL {X  -162.820, Y  +399.588, Z    +0.000, E1   +70.462, E3 +146520.432}
SPL {X  -159.703, Y  +348.793, Z    +0.000, E1   +73.194, E3 +146527.736}
SPL {X  -158.911, Y  +345.038, Z    +0.000, E1   +72.209, E3 +146539.953}
SPL {X  -157.738, Y  +340.137, Z    +0.000, E1   +71.006, E3 +146554.769}
SPL {X  -155.731, Y  +332.978, Z    +0.000, E1   +69.670, E3 +146571.419}
SPL {X  -153.052, Y  +324.954, Z    +0.000, E1   +68.671, E3 +146585.381}
SPL {X  -148.581, Y  +313.911, Z    +0.000, E1   +68.095, E3 +146598.171}
SPL {X  -143.686, Y  +303.920, Z    +0.000, E1   +67.419, E3 +146610.308}
SPL {X  -138.888, Y  +295.526, Z    +0.000, E1   +66.767, E3 +146620.643}
SPL {X  -134.802, Y  +289.183, Z    +0.000, E1   +66.143, E3 +146628.767}
SPL {X  -131.727, Y  +284.801, Z    +0.000, E1   +65.590, E3 +146634.781}
SPL {X  -128.890, Y  +281.012, Z    +0.000, E1   +65.392, E3 +146638.526}
SPL {X  -121.325, Y  +271.915, Z    +0.000, E1   +67.092, E3 +146638.092}
SPL {X   -79.997, Y  +238.687, Z    +0.000, E1   +54.340, E3 +146796.848}
ENDSPLINE

SPLINE
SPL {X  -139.099, Y  +295.872, Z    +0.000, E1   +47.860, E3 +146924.724}
SPL {X  -156.463, Y  +335.448, Z    +0.000, E1   +33.333, E3 +146935.432}
SPL {X  -161.312, Y  +358.394, Z    +0.000, E1   +19.478, E3 +146937.067}
SPL {X  -162.549, Y  +371.111, Z    +0.000, E1    +9.905, E3 +146937.127}
SPL {X  -162.818, Y  +379.769, Z    +0.000, E1    +2.607, E3 +146936.869}
SPL {X  -162.820, Y  +382.500, Z    +0.000, E1    +0.000, E3 +146936.438}
SPL {X  -162.820, Y  +384.989, Z    +0.000, E1    -3.865, E3 +146936.165}
SPL {X  -162.820, Y  +391.404, Z    +0.000, E1   -16.767, E3 +146936.012}
SPL {X  -162.820, Y  +397.742, Z    +0.000, E1   -30.068, E3 +146936.078}
SPL {X  -162.820, Y  +403.938, Z    +0.000, E1   -41.112, E3 +146936.057}
SPL {X  -162.820, Y  +415.430, Z    +0.000, E1   -55.307, E3 +146936.256}
SPL {X  -162.820, Y  +466.986, Z    +0.000, E1   -71.397, E3 +146948.016}
SPL {X  -162.820, Y  +661.594, Z    +0.000, E1   -73.988, E3 +147033.642}
ENDSPLINE

SPLINE
SPL {X  -162.820, Y  +634.363, Z    +0.000, E1   -70.793, E3 +147047.220}
ENDSPLINE

SPLINE
SPL {X  -162.820, Y  +649.777, Z    +0.000, E1   -70.953, E3 +147056.979}
SPL {X  -162.820, Y  +667.477, Z    +0.000, E1   -70.889, E3 +147070.287}
SPL {X  -162.097, Y  +688.831, Z    +0.000, E1   -70.910, E3 +147085.658}
SPL {X  -159.319, Y  +707.081, Z    +0.000, E1   -70.563, E3 +147101.944}
SPL {X  -156.566, Y  +718.194, Z    +0.000, E1   -70.115, E3 +147113.749}
SPL {X  -153.268, Y  +728.449, Z    +0.000, E1   -69.855, E3 +147123.374}
SPL {X  -150.033, Y  +736.750, Z    +0.000, E1   -69.498, E3 +147132.086}
SPL {X  -146.704, Y  +744.128, Z    +0.000, E1   -68.985, E3 +147141.208}
SPL {X  -142.102, Y  +752.982, Z    +0.000, E1   -68.357, E3 +147151.946}
SPL {X  -138.073, Y  +759.791, Z    +0.000, E1   -67.958, E3 +147159.116}
SPL {X  -134.977, Y  +764.558, Z    +0.000, E1   -67.353, E3 +147166.037}
SPL {X  -130.728, Y  +770.560, Z    +0.000, E1   -66.612, E3 +147174.072}
SPL {X  -125.283, Y  +777.493, Z    +0.000, E1   -66.879, E3 +147177.798}
SPL {X   -78.323, Y  +816.244, Z    +0.000, E1   -56.979, E3 +147284.893}
ENDSPLINE

SPLINE
SPL {X   -93.623, Y  +806.710, Z    +0.000, E1   -55.511, E3 +147430.579}
SPL {X  -138.493, Y  +759.115, Z    +0.000, E1   -50.023, E3 +147478.408}
SPL {X  -149.871, Y  +737.133, Z    +0.000, E1   -43.112, E3 +147483.822}
SPL {X  -157.876, Y  +713.320, Z    +0.000, E1   -31.448, E3 +147483.597}
SPL {X  -161.323, Y  +695.531, Z    +0.000, E1   -20.168, E3 +147485.641}
SPL {X  -162.428, Y  +684.786, Z    +0.000, E1   -11.829, E3 +147485.538}
SPL {X  -162.809, Y  +675.372, Z    +0.000, E1    -3.788, E3 +147485.652}
SPL {X  -162.820, Y  +671.476, Z    +0.000, E1    +0.020, E3 +147485.165}
SPL {X  -162.820, Y  +668.959, Z    +0.000, E1    +4.387, E3 +147484.886}
SPL {X  -162.820, Y  +664.344, Z    +0.000, E1   +14.120, E3 +147484.785}
SPL {X  -162.820, Y  +658.993, Z    +0.000, E1   +25.845, E3 +147484.875}
SPL {X  -162.820, Y  +650.479, Z    +0.000, E1   +41.861, E3 +147485.034}
SPL {X  -162.820, Y  +634.626, Z    +0.000, E1   +60.916, E3 +147484.318}
SPL {X  -162.820, Y  +600.578, Z    +0.000, E1   +80.831, E3 +147474.975}
SPL {X  -162.820, Y  +567.495, Z    +0.000, E1   +70.620, E3 +147510.100}
SPL {X  -162.820, Y  +416.506, Z    +0.000, E1   +71.398, E3 +147594.446}
SPL {X  -162.820, Y  +411.010, Z    +0.000, E1   +70.614, E3 +147605.897}
SPL {X  -162.820, Y  +391.151, Z    +0.000, E1   +70.927, E3 +147617.351}
SPL {X  -159.025, Y  +345.550, Z    +0.000, E1   +73.389, E3 +147623.032}
ENDSPLINE

SPLINE
SPL {X  -159.121, Y  +345.992, Z    +0.000, E1   +72.455, E3 +147631.999}
ENDSPLINE

SPLINE
SPL {X  -158.667, Y  +343.959, Z    +0.000, E1   +71.763, E3 +147640.107}
SPL {X  -157.901, Y  +340.780, Z    +0.000, E1   +71.006, E3 +147649.215}
SPL {X  -156.755, Y  +336.473, Z    +0.000, E1   +70.264, E3 +147658.922}
SPL {X  -155.322, Y  +331.660, Z    +0.000, E1   +69.461, E3 +147669.169}
SPL {X  -154.241, Y  +328.346, Z    +0.000, E1   +68.710, E3 +147677.600}
SPL {X  -151.364, Y  +320.507, Z    +0.000, E1   +68.513, E3 +147685.226}
SPL {X  -147.865, Y  +312.336, Z    +0.000, E1   +67.945, E3 +147695.516}
SPL {X  -143.686, Y  +303.920, Z    +0.000, E1   +67.419, E3 +147705.546}
SPL {X  -138.888, Y  +295.526, Z    +0.000, E1   +66.767, E3 +147715.881}
SPL {X  -134.802, Y  +289.183, Z    +0.000, E1   +66.143, E3 +147724.005}
SPL {X  -131.727, Y  +284.801, Z    +0.000, E1   +65.590, E3 +147730.019}
SPL {X  -128.890, Y  +281.012, Z    +0.000, E1   +65.392, E3 +147733.764}
SPL {X  -121.325, Y  +271.915, Z    +0.000, E1   +67.092, E3 +147733.330}
SPL {X   -79.997, Y  +238.687, Z    +0.000, E1   +54.340, E3 +147892.087}
ENDSPLINE

SPLINE
SPL {X  -139.099, Y  +295.872, Z    +0.000, E1   +47.860, E3 +148019.962}
SPL {X  -156.463, Y  +335.448, Z    +0.000, E1   +33.333, E3 +148030.670}
SPL {X  -161.312, Y  +358.394, Z    +0.000, E1   +19.478, E3 +148032.305}
SPL {X  -162.549, Y  +371.111, Z    +0.000, E1    +9.905, E3 +148032.365}
SPL {X  -162.818, Y  +379.769, Z    +0.000, E1    +2.607, E3 +148032.107}
SPL {X  -162.820, Y  +382.897, Z    +0.000, E1    -0.379, E3 +148031.591}
SPL {X  -162.820, Y  +387.689, Z    +0.000, E1    -9.147, E3 +148031.310}
SPL {X  -162.820, Y  +392.805, Z    +0.000, E1   -19.930, E3 +148031.283}
SPL {X  -162.820, Y  +397.742, Z    +0.000, E1   -30.068, E3 +148031.316}
SPL {X  -162.820, Y  +403.938, Z    +0.000, E1   -41.112, E3 +148031.295}
SPL {X  -162.820, Y  +415.430, Z    +0.000, E1   -55.307, E3 +148031.494}
SPL {X  -162.820, Y  +466.986, Z    +0.000, E1   -71.397, E3 +148043.254}
SPL {X  -162.820, Y  +661.594, Z    +0.000, E1   -73.988, E3 +148128.880}
ENDSPLINE

SPLINE
SPL {X  -162.820, Y  +634.363, Z    +0.000, E1   -70.793, E3 +148142.458}
ENDSPLINE

SPLINE
SPL {X  -162.820, Y  +649.777, Z    +0.000, E1   -70.953, E3 +148152.217}
SPL {X  -162.820, Y  +667.477, Z    +0.000, E1   -70.889, E3 +148165.525}
SPL {X  -162.462, Y  +684.286, Z    +0.000, E1   -70.880, E3 +148177.758}
SPL {X  -160.799, Y  +699.074, Z    +0.000, E1   -70.750, E3 +148189.623}
SPL {X  -158.733, Y  +709.754, Z    +0.000, E1   -70.504, E3 +148199.505}
SPL {X  -156.566, Y  +718.194, Z    +0.000, E1   -70.115, E3 +148208.987}
SPL {X  -153.268, Y  +728.449, Z    +0.000, E1   -69.855, E3 +148218.612}
SPL {X  -150.033, Y  +736.750, Z    +0.000, E1   -69.498, E3 +148227.324}
SPL {X  -146.704, Y  +744.128, Z    +0.000, E1   -68.985, E3 +148236.446}
SPL {X  -143.061, Y  +751.243, Z    +0.000, E1   -68.459, E3 +148245.142}
SPL {X  -139.143, Y  +758.055, Z    +0.000, E1   -68.038, E3 +148252.704}
SPL {X  -136.095, Y  +762.879, Z    +0.000, E1   -67.470, E3 +148259.339}
SPL {X  -133.055, Y  +767.344, Z    +0.000, E1   -67.024, E3 +148264.970}
SPL {X  -129.955, Y  +771.593, Z    +0.000, E1   -66.476, E3 +148270.611}
SPL {X  -125.283, Y  +777.493, Z    +0.000, E1   -66.879, E3 +148273.036}
SPL {X   -78.323, Y  +816.244, Z    +0.000, E1   -56.979, E3 +148380.131}
ENDSPLINE

SPLINE
SPL {X   -93.623, Y  +806.710, Z    +0.000, E1   -55.511, E3 +148525.818}
SPL {X  -138.493, Y  +759.115, Z    +0.000, E1   -50.023, E3 +148573.646}
SPL {X  -149.871, Y  +737.133, Z    +0.000, E1   -43.112, E3 +148579.060}
SPL {X  -157.876, Y  +713.320, Z    +0.000, E1   -31.448, E3 +148578.835}
SPL {X  -161.323, Y  +695.531, Z    +0.000, E1   -20.168, E3 +148580.879}
SPL {X  -162.626, Y  +681.447, Z    +0.000, E1    -9.120, E3 +148580.868}
SPL {X  -162.820, Y  +673.597, Z    +0.000, E1    -2.055, E3 +148580.861}
SPL {X  -162.820, Y  +671.476, Z    +0.000, E1    +0.020, E3 +148580.404}
SPL {X  -162.820, Y  +668.959, Z    +0.000, E1    +4.387, E3 +148580.124}
SPL {X  -162.820, Y  +664.344, Z    +0.000, E1   +14.120, E3 +148580.023}
SPL {X  -162.820, Y  +658.993, Z    +0.000, E1   +25.845, E3 +148580.113}
SPL {X  -162.820, Y  +652.443, Z    +0.000, E1   +38.206, E3 +148580.849}
SPL {X  -162.820, Y  +640.832, Z    +0.000, E1   +55.385, E3 +148579.562}
SPL {X  -162.820, Y  +625.562, Z    +0.000, E1   +67.658, E3 +148578.616}
SPL {X  -162.820, Y  +600.578, Z    +0.000, E1   +80.831, E3 +148570.213}
SPL {X  -162.820, Y  +567.495, Z    +0.000, E1   +70.620, E3 +148605.338}
SPL {X  -162.820, Y  +416.506, Z    +0.000, E1   +71.398, E3 +148689.684}
SPL {X  -162.820, Y  +411.010, Z    +0.000, E1   +70.614, E3 +148701.135}
SPL {X  -162.820, Y  +399.588, Z    +0.000, E1   +70.462, E3 +148710.908}
SPL {X  -159.703, Y  +348.793, Z    +0.000, E1   +73.194, E3 +148718.213}
SPL {X  -159.121, Y  +345.992, Z    +0.000, E1   +72.455, E3 +148727.237}
SPL {X  -158.667, Y  +343.959, Z    +0.000, E1   +71.763, E3 +148735.345}
SPL {X  -157.901, Y  +340.780, Z    +0.000, E1   +71.006, E3 +148744.453}
SPL {X  -156.755, Y  +336.473, Z    +0.000, E1   +70.264, E3 +148754.161}
SPL {X  -155.322, Y  +331.660, Z    +0.000, E1   +69.461, E3 +148764.407}
SPL {X  -154.241, Y  +328.346, Z    +0.000, E1   +68.710, E3 +148772.838}
SPL {X  -151.364, Y  +320.507, Z    +0.000, E1   +68.513, E3 +148780.464}
SPL {X  -147.865, Y  +312.336, Z    +0.000, E1   +67.945, E3 +148790.754}
SPL {X  -144.739, Y  +305.928, Z    +0.000, E1   +67.540, E3 +148798.337}
SPL {X  -141.308, Y  +299.614, Z    +0.000, E1   +67.079, E3 +148806.128}
SPL {X  -137.907, Y  +293.943, Z    +0.000, E1   +66.608, E3 +148813.107}
SPL {X  -134.802, Y  +289.183, Z    +0.000, E1   +66.143, E3 +148819.243}
SPL {X  -131.727, Y  +284.801, Z    +0.000, E1   +65.590, E3 +148825.257}
SPL {X  -128.890, Y  +281.012, Z    +0.000, E1   +65.392, E3 +148829.003}
SPL {X  -121.325, Y  +271.915, Z    +0.000, E1   +67.092, E3 +148828.568}
SPL {X   -79.997, Y  +238.687, Z    +0.000, E1   +54.340, E3 +148987.325}
ENDSPLINE

SPLINE
SPL {X  -139.099, Y  +295.872, Z    +0.000, E1   +47.860, E3 +149115.200}
SPL {X  -156.463, Y  +335.448, Z    +0.000, E1   +33.333, E3 +149125.908}
SPL {X  -161.312, Y  +358.394, Z    +0.000, E1   +19.478, E3 +149127.543}
SPL {X  -162.549, Y  +371.111, Z    +0.000, E1    +9.905, E3 +149127.603}
SPL {X  -162.818, Y  +379.769, Z    +0.000, E1    +2.607, E3 +149127.345}
SPL {X  -162.820, Y  +382.500, Z    +0.000, E1    +0.000, E3 +149126.914}
SPL {X  -162.820, Y  +384.989, Z    +0.000, E1    -3.865, E3 +149126.641}
SPL {X  -162.820, Y  +391.404, Z    +0.000, E1   -16.767, E3 +149126.488}
SPL {X  -162.820, Y  +397.742, Z    +0.000, E1   -30.068, E3 +149126.554}
SPL {X  -162.820, Y  +403.938, Z    +0.000, E1   -41.112, E3 +149126.533}
SPL {X  -162.820, Y  +415.430, Z    +0.000, E1   -55.307, E3 +149126.732}
SPL {X  -162.820, Y  +466.986, Z    +0.000, E1   -71.397, E3 +149138.492}
SPL {X  -162.820, Y  +661.594, Z    +0.000, E1   -73.988, E3 +149224.118}
ENDSPLINE

SPLINE
SPL {X  -162.820, Y  +634.363, Z    +0.000, E1   -70.793, E3 +149237.696}
ENDSPLINE

SPLINE
SPL {X  -162.820, Y  +649.777, Z    +0.000, E1   -70.953, E3 +149247.455}
SPL {X  -162.820, Y  +667.477, Z    +0.000, E1   -70.889, E3 +149260.763}
SPL {X  -162.462, Y  +684.286, Z    +0.000, E1   -70.880, E3 +149272.997}
SPL {X  -160.799, Y  +699.074, Z    +0.000, E1   -70.750, E3 +149284.861}
SPL {X  -158.733, Y  +709.754, Z    +0.000, E1   -70.504, E3 +149294.743}
SPL {X  -156.566, Y  +718.194, Z    +0.000, E1   -70.115, E3 +149304.225}
SPL {X  -153.268, Y  +728.449, Z    +0.000, E1   -69.855, E3 +149313.850}
SPL {X  -150.033, Y  +736.750, Z    +0.000, E1   -69.498, E3 +149322.562}
SPL {X  -146.704, Y  +744.128, Z    +0.000, E1   -68.985, E3 +149331.684}
SPL {X  -143.061, Y  +751.243, Z    +0.000, E1   -68.459, E3 +149340.380}
SPL {X  -139.143, Y  +758.055, Z    +0.000, E1   -68.038, E3 +149347.942}
SPL {X  -134.977, Y  +764.558, Z    +0.000, E1   -67.353, E3 +149356.513}
SPL {X  -130.728, Y  +770.560, Z    +0.000, E1   -66.612, E3 +149364.549}
SPL {X  -127.384, Y  +774.909, Z    +0.000, E1   -66.413, E3 +149368.491}
SPL {X  -122.177, Y  +781.125, Z    +0.000, E1   -67.611, E3 +149367.860}
SPL {X   -78.323, Y  +816.244, Z    +0.000, E1   -56.979, E3 +149475.369}
ENDSPLINE

SPLINE
SPL {X   -93.623, Y  +806.710, Z    +0.000, E1   -55.511, E3 +149621.056}
SPL {X  -143.027, Y  +751.304, Z    +0.000, E1   -47.932, E3 +149671.116}
SPL {X  -157.876, Y  +713.320, Z    +0.000, E1   -31.448, E3 +149674.073}
SPL {X  -161.323, Y  +695.531, Z    +0.000, E1   -20.168, E3 +149676.117}
SPL {X  -162.428, Y  +684.786, Z    +0.000, E1   -11.829, E3 +149676.014}
SPL {X  -162.809, Y  +675.372, Z    +0.000, E1    -3.788, E3 +149676.128}
SPL {X  -162.820, Y  +671.476, Z    +0.000, E1    +0.020, E3 +149675.642}
SPL {X  -162.820, Y  +668.959, Z    +0.000, E1    +4.387, E3 +149675.362}
SPL {X  -162.820, Y  +664.344, Z    +0.000, E1   +14.120, E3 +149675.261}
SPL {X  -162.820, Y  +658.993, Z    +0.000, E1   +25.845, E3 +149675.351}
SPL {X  -162.820, Y  +652.443, Z    +0.000, E1   +38.206, E3 +149676.087}
SPL {X  -162.820, Y  +640.832, Z    +0.000, E1   +55.385, E3 +149674.800}
SPL {X  -162.820, Y  +625.562, Z    +0.000, E1   +67.658, E3 +149673.854}
SPL {X  -162.820, Y  +600.578, Z    +0.000, E1   +80.831, E3 +149665.452}
SPL {X  -162.820, Y  +567.495, Z    +0.000, E1   +70.620, E3 +149700.576}
SPL {X  -162.820, Y  +416.506, Z    +0.000, E1   +71.398, E3 +149784.922}
SPL {X  -162.820, Y  +411.010, Z    +0.000, E1   +70.614, E3 +149796.373}
SPL {X  -162.820, Y  +399.588, Z    +0.000, E1   +70.462, E3 +149806.146}
SPL {X  -159.703, Y  +348.793, Z    +0.000, E1   +73.194, E3 +149813.451}
SPL {X  -158.911, Y  +345.038, Z    +0.000, E1   +72.209, E3 +149825.667}
SPL {X  -158.117, Y  +341.649, Z    +0.000, E1   +71.181, E3 +149837.623}
SPL {X  -156.755, Y  +336.473, Z    +0.000, E1   +70.264, E3 +149849.399}
SPL {X  -155.322, Y  +331.660, Z    +0.000, E1   +69.461, E3 +149859.645}
SPL {X  -154.241, Y  +328.346, Z    +0.000, E1   +68.710, E3 +149868.076}
SPL {X  -151.364, Y  +320.507, Z    +0.000, E1   +68.513, E3 +149875.702}
SPL {X  -147.865, Y  +312.336, Z    +0.000, E1   +67.945, E3 +149885.992}
SPL {X  -143.686, Y  +303.920, Z    +0.000, E1   +67.419, E3 +149896.023}
SPL {X  -138.888, Y  +295.526, Z    +0.000, E1   +66.767, E3 +149906.357}
SPL {X  -134.802, Y  +289.183, Z    +0.000, E1   +66.143, E3 +149914.481}
SPL {X  -131.727, Y  +284.801, Z    +0.000, E1   +65.590, E3 +149920.495}
SPL {X  -128.890, Y  +281.012, Z    +0.000, E1   +65.392, E3 +149924.241}
SPL {X  -121.325, Y  +271.915, Z    +0.000, E1   +67.092, E3 +149923.806}
SPL {X   -79.997, Y  +238.687, Z    +0.000, E1   +54.340, E3 +150082.563}
ENDSPLINE

SPLINE
SPL {X  -139.099, Y  +295.872, Z    +0.000, E1   +47.860, E3 +150210.438}
SPL {X  -156.463, Y  +335.448, Z    +0.000, E1   +33.333, E3 +150221.147}
SPL {X  -161.312, Y  +358.394, Z    +0.000, E1   +19.478, E3 +150222.781}
SPL {X  -162.549, Y  +371.111, Z    +0.000, E1    +9.905, E3 +150222.841}
SPL {X  -162.818, Y  +379.769, Z    +0.000, E1    +2.607, E3 +150222.583}
SPL {X  -162.820, Y  +382.500, Z    +0.000, E1    +0.000, E3 +150222.152}
SPL {X  -162.820, Y  +383.721, Z    +0.000, E1    -1.897, E3 +150221.890}
SPL {X  -162.820, Y  +387.689, Z    +0.000, E1    -9.147, E3 +150221.786}
SPL {X  -162.820, Y  +392.805, Z    +0.000, E1   -19.930, E3 +150221.760}
SPL {X  -162.820, Y  +397.742, Z    +0.000, E1   -30.068, E3 +150221.792}
SPL {X  -162.820, Y  +403.938, Z    +0.000, E1   -41.112, E3 +150221.771}
SPL {X  -162.820, Y  +415.430, Z    +0.000, E1   -55.307, E3 +150221.970}
SPL {X  -162.820, Y  +466.986, Z    +0.000, E1   -71.397, E3 +150233.730}
SPL {X  -162.820, Y  +661.594, Z    +0.000, E1   -73.988, E3 +150319.356}
ENDSPLINE

SPLINE
SPL {X  -162.820, Y  +646.360, Z    +0.000, E1   -70.938, E3 +150340.487}
ENDSPLINE

SPLINE
SPL {X  -162.820, Y  +667.477, Z    +0.000, E1   -70.889, E3 +150356.002}
SPL {X  -162.462, Y  +684.286, Z    +0.000, E1   -70.880, E3 +150368.235}
SPL {X  -160.799, Y  +699.074, Z    +0.000, E1   -70.750, E3 +150380.099}
SPL {X  -158.733, Y  +709.754, Z    +0.000, E1   -70.504, E3 +150389.982}
SPL {X  -156.566, Y  +718.194, Z    +0.000, E1   -70.115, E3 +150399.463}
SPL {X  -153.268, Y  +728.449, Z    +0.000, E1   -69.855, E3 +150409.088}
SPL {X  -150.033, Y  +736.750, Z    +0.000, E1   -69.498, E3 +150417.800}
SPL {X  -146.704, Y  +744.128, Z    +0.000, E1   -68.985, E3 +150426.922}
SPL {X  -143.061, Y  +751.243, Z    +0.000, E1   -68.459, E3 +150435.618}
SPL {X  -139.143, Y  +758.055, Z    +0.000, E1   -68.038, E3 +150443.180}
SPL {X  -134.977, Y  +764.558, Z    +0.000, E1   -67.353, E3 +150451.751}
SPL {X  -130.728, Y  +770.560, Z    +0.000, E1   -66.612, E3 +150459.787}
SPL {X  -127.384, Y  +774.909, Z    +0.000, E1   -66.413, E3 +150463.729}
SPL {X  -122.177, Y  +781.125, Z    +0.000, E1   -67.611, E3 +150463.098}
SPL {X   -78.323, Y  +816.244, Z    +0.000, E1   -56.979, E3 +150570.607}
ENDSPLINE

SPLINE
SPL {X   -93.623, Y  +806.710, Z    +0.000, E1   -55.511, E3 +150716.294}
SPL {X  -143.027, Y  +751.304, Z    +0.000, E1   -47.932, E3 +150766.354}
SPL {X  -157.876, Y  +713.320, Z    +0.000, E1   -31.448, E3 +150769.311}
SPL {X  -161.323, Y  +695.531, Z    +0.000, E1   -20.168, E3 +150771.355}
SPL {X  -162.428, Y  +684.786, Z    +0.000, E1   -11.829, E3 +150771.252}
SPL {X  -162.809, Y  +675.372, Z    +0.000, E1    -3.788, E3 +150771.367}
SPL {X  -162.820, Y  +671.476, Z    +0.000, E1    +0.020, E3 +150770.880}
SPL {X  -162.820, Y  +668.959, Z    +0.000, E1    +4.387, E3 +150770.601}
SPL {X  -162.820, Y  +664.344, Z    +0.000, E1   +14.120, E3 +150770.499}
SPL {X  -162.820, Y  +658.993, Z    +0.000, E1   +25.845, E3 +150770.589}
SPL {X  -162.820, Y  +652.443, Z    +0.000, E1   +38.206, E3 +150771.325}
SPL {X  -162.820, Y  +640.832, Z    +0.000, E1   +55.385, E3 +150770.038}
SPL {X  -162.820, Y  +625.562, Z    +0.000, E1   +67.658, E3 +150769.092}
SPL {X  -162.820, Y  +600.578, Z    +0.000, E1   +80.831, E3 +150760.690}
SPL {X  -162.820, Y  +567.495, Z    +0.000, E1   +70.620, E3 +150795.814}
SPL {X  -162.820, Y  +416.506, Z    +0.000, E1   +71.398, E3 +150880.160}
SPL {X  -162.820, Y  +411.010, Z    +0.000, E1   +70.614, E3 +150891.611}
SPL {X  -162.820, Y  +399.588, Z    +0.000, E1   +70.462, E3 +150901.384}
SPL {X  -159.703, Y  +348.793, Z    +0.000, E1   +73.194, E3 +150908.689}
SPL {X  -158.911, Y  +345.038, Z    +0.000, E1   +72.209, E3 +150920.905}
SPL {X  -158.117, Y  +341.649, Z    +0.000, E1   +71.181, E3 +150932.861}
SPL {X  -156.755, Y  +336.473, Z    +0.000, E1   +70.264, E3 +150944.637}
SPL {X  -155.322, Y  +331.660, Z    +0.000, E1   +69.461, E3 +150954.883}
SPL {X  -153.052, Y  +324.954, Z    +0.000, E1   +68.671, E3 +150966.334}
SPL {X  -149.405, Y  +315.782, Z    +0.000, E1   +68.161, E3 +150977.099}
SPL {X  -145.408, Y  +307.240, Z    +0.000, E1   +67.667, E3 +150987.078}
SPL {X  -141.308, Y  +299.614, Z    +0.000, E1   +67.079, E3 +150996.604}
SPL {X  -137.907, Y  +293.943, Z    +0.000, E1   +66.608, E3 +151003.583}
SPL {X  -134.802, Y  +289.183, Z    +0.000, E1   +66.143, E3 +151009.719}
SPL {X  -131.727, Y  +284.801, Z    +0.000, E1   +65.590, E3 +151015.733}
SPL {X  -128.890, Y  +281.012, Z    +0.000, E1   +65.392, E3 +151019.479}
SPL {X  -121.325, Y  +271.915, Z    +0.000, E1   +67.092, E3 +151019.045}
SPL {X   -79.997, Y  +238.687, Z    +0.000, E1   +54.340, E3 +151177.801}
ENDSPLINE

SPLINE
SPL {X  -139.099, Y  +295.872, Z    +0.000, E1   +47.860, E3 +151305.676}
SPL {X  -156.463, Y  +335.448, Z    +0.000, E1   +33.333, E3 +151316.385}
SPL {X  -161.312, Y  +358.394, Z    +0.000, E1   +19.478, E3 +151318.019}
SPL {X  -162.549, Y  +371.111, Z    +0.000, E1    +9.905, E3 +151318.079}
SPL {X  -162.818, Y  +379.769, Z    +0.000, E1    +2.607, E3 +151317.821}
SPL {X  -162.820, Y  +382.500, Z    +0.000, E1    +0.000, E3 +151317.391}
SPL {X  -162.820, Y  +383.721, Z    +0.000, E1    -1.897, E3 +151317.128}
SPL {X  -162.820, Y  +387.689, Z    +0.000, E1    -9.147, E3 +151317.024}
SPL {X  -162.820, Y  +392.805, Z    +0.000, E1   -19.930, E3 +151316.998}
SPL {X  -162.820, Y  +397.742, Z    +0.000, E1   -30.068, E3 +151317.030}
SPL {X  -162.820, Y  +403.938, Z    +0.000, E1   -41.112, E3 +151317.009}
SPL {X  -162.820, Y  +415.430, Z    +0.000, E1   -55.307, E3 +151317.209}
SPL {X  -162.820, Y  +466.986, Z    +0.000, E1   -71.397, E3 +151328.968}
SPL {X  -162.820, Y  +661.594, Z    +0.000, E1   -73.988, E3 +151414.594}
ENDSPLINE

SPLINE
SPL {X  -162.820, Y  +646.360, Z    +0.000, E1   -70.938, E3 +151435.725}
ENDSPLINE

SPLINE
SPL {X  -162.820, Y  +667.477, Z    +0.000, E1   -70.889, E3 +151451.240}
SPL {X  -162.462, Y  +684.286, Z    +0.000, E1   -70.880, E3 +151463.473}
SPL {X  -160.799, Y  +699.074, Z    +0.000, E1   -70.750, E3 +151475.337}
SPL {X  -158.733, Y  +709.754, Z    +0.000, E1   -70.504, E3 +151485.220}
SPL {X  -156.566, Y  +718.194, Z    +0.000, E1   -70.115, E3 +151494.701}
SPL {X  -153.268, Y  +728.449, Z    +0.000, E1   -69.855, E3 +151504.327}
SPL {X  -150.033, Y  +736.750, Z    +0.000, E1   -69.498, E3 +151513.038}
SPL {X  -146.704, Y  +744.128, Z    +0.000, E1   -68.985, E3 +151522.160}
SPL {X  -143.061, Y  +751.243, Z    +0.000, E1   -68.459, E3 +151530.856}
SPL {X  -139.143, Y  +758.055, Z    +0.000, E1   -68.038, E3 +151538.418}
SPL {X  -134.977, Y  +764.558, Z    +0.000, E1   -67.353, E3 +151546.990}
SPL {X  -130.728, Y  +770.560, Z    +0.000, E1   -66.612, E3 +151555.025}
SPL {X  -125.283, Y  +777.493, Z    +0.000, E1   -66.879, E3 +151558.750}
SPL {X   -78.323, Y  +816.244, Z    +0.000, E1   -56.979, E3 +151665.845}
ENDSPLINE

SPLINE
SPL {X   -93.623, Y  +806.710, Z    +0.000, E1   -55.511, E3 +151811.532}
SPL {X  -138.493, Y  +759.115, Z    +0.000, E1   -50.023, E3 +151859.360}
SPL {X  -149.871, Y  +737.133, Z    +0.000, E1   -43.112, E3 +151864.774}
SPL {X  -157.876, Y  +713.320, Z    +0.000, E1   -31.448, E3 +151864.550}
SPL {X  -161.323, Y  +695.531, Z    +0.000, E1   -20.168, E3 +151866.593}
SPL {X  -162.428, Y  +684.786, Z    +0.000, E1   -11.829, E3 +151866.490}
SPL {X  -162.809, Y  +675.372, Z    +0.000, E1    -3.788, E3 +151866.605}
SPL {X  -162.820, Y  +671.476, Z    +0.000, E1    +0.020, E3 +151866.118}
SPL {X  -162.820, Y  +668.959, Z    +0.000, E1    +4.387, E3 +151865.839}
SPL {X  -162.820, Y  +664.344, Z    +0.000, E1   +14.120, E3 +151865.738}
SPL {X  -162.820, Y  +658.993, Z    +0.000, E1   +25.845, E3 +151865.827}
SPL {X  -162.820, Y  +650.479, Z    +0.000, E1   +41.861, E3 +151865.987}
SPL {X  -162.820, Y  +634.626, Z    +0.000, E1   +60.916, E3 +151865.270}
SPL {X  -162.820, Y  +600.578, Z    +0.000, E1   +80.831, E3 +151855.928}
SPL {X  -162.820, Y  +567.495, Z    +0.000, E1   +70.620, E3 +151891.052}
SPL {X  -162.820, Y  +416.506, Z    +0.000, E1   +71.398, E3 +151975.398}
SPL {X  -162.820, Y  +411.010, Z    +0.000, E1   +70.614, E3 +151986.849}
SPL {X  -162.820, Y  +399.588, Z    +0.000, E1   +70.462, E3 +151996.623}
SPL {X  -159.703, Y  +348.793, Z    +0.000, E1   +73.194, E3 +152003.927}
SPL {X  -158.911, Y  +345.038, Z    +0.000, E1   +72.209, E3 +152016.143}
SPL {X  -158.117, Y  +341.649, Z    +0.000, E1   +71.181, E3 +152028.099}
SPL {X  -156.755, Y  +336.473, Z    +0.000, E1   +70.264, E3 +152039.875}
SPL {X  -155.322, Y  +331.660, Z    +0.000, E1   +69.461, E3 +152050.121}
ENDSPLINE

SPLINE
SPL {X  -156.716, Y  +336.338, Z    +0.000, E1   +67.007, E3 +152066.057}
ENDSPLINE

SPLINE
SPL {X  -153.279, Y  +325.584, Z    +0.000, E1   +66.662, E3 +152077.672}
SPL {X  -149.546, Y  +316.107, Z    +0.000, E1   +66.216, E3 +152088.848}
SPL {X  -147.033, Y  +310.560, Z    +0.000, E1   +65.497, E3 +152098.062}
SPL {X  -144.094, Y  +304.689, Z    +0.000, E1   +65.338, E3 +152104.074}
SPL {X  -141.093, Y  +299.241, Z    +0.000, E1   +65.039, E3 +152110.386}
SPL {X  -138.425, Y  +294.774, Z    +0.000, E1   +64.416, E3 +152117.570}
SPL {X  -134.374, Y  +288.555, Z    +0.000, E1   +63.758, E3 +152126.212}
SPL {X  -128.896, Y  +281.020, Z    +0.000, E1   +64.005, E3 +152131.335}
SPL {X   -85.291, Y  +241.807, Z    +0.000, E1   +53.957, E3 +152276.743}
ENDSPLINE

SPLINE
SPL {X  -136.861, Y  +292.299, Z    +0.000, E1   +47.815, E3 +152404.364}
SPL {X  -156.420, Y  +335.300, Z    +0.000, E1   +31.885, E3 +152412.153}
SPL {X  -161.293, Y  +358.252, Z    +0.000, E1   +18.542, E3 +152413.871}
SPL {X  -162.487, Y  +370.094, Z    +0.000, E1   +10.144, E3 +152413.949}
SPL {X  -162.818, Y  +379.612, Z    +0.000, E1    +2.663, E3 +152413.925}
SPL {X  -162.820, Y  +382.500, Z    +0.000, E1    +0.000, E3 +152413.518}
SPL {X  -162.820, Y  +383.629, Z    +0.000, E1    -1.565, E3 +152413.211}
SPL {X  -162.820, Y  +387.649, Z    +0.000, E1    -8.215, E3 +152413.199}
SPL {X  -162.820, Y  +392.460, Z    +0.000, E1   -17.627, E3 +152413.181}
SPL {X  -162.820, Y  +397.383, Z    +0.000, E1   -27.100, E3 +152413.251}
SPL {X  -162.820, Y  +404.822, Z    +0.000, E1   -40.113, E3 +152412.902}
SPL {X  -162.820, Y  +416.103, Z    +0.000, E1   -54.033, E3 +152412.754}
SPL {X  -162.820, Y  +472.592, Z    +0.000, E1   -70.190, E3 +152428.356}
SPL {X  -162.820, Y  +605.049, Z    +0.000, E1   -68.347, E3 +152522.838}
SPL {X  -162.820, Y  +616.480, Z    +0.000, E1   -67.752, E3 +152537.531}
SPL {X  -162.820, Y  +631.154, Z    +0.000, E1   -67.735, E3 +152550.066}
SPL {X  -162.820, Y  +647.590, Z    +0.000, E1   -67.861, E3 +152563.101}
SPL {X  -162.820, Y  +663.021, Z    +0.000, E1   -67.764, E3 +152576.938}
SPL {X  -162.642, Y  +681.112, Z    +0.000, E1   -67.812, E3 +152592.090}
SPL {X  -161.154, Y  +696.734, Z    +0.000, E1   -67.591, E3 +152607.087}
SPL {X  -158.503, Y  +710.744, Z    +0.000, E1   -67.284, E3 +152621.618}
SPL {X  -155.060, Y  +723.165, Z    +0.000, E1   -66.797, E3 +152635.794}
SPL {X  -151.511, Y  +733.123, Z    +0.000, E1   -66.286, E3 +152647.948}
SPL {X  -147.735, Y  +741.944, Z    +0.000, E1   -65.827, E3 +152658.474}
SPL {X  -144.196, Y  +749.116, Z    +0.000, E1   -65.203, E3 +152668.474}
SPL {X  -139.960, Y  +756.696, Z    +0.000, E1   -64.606, E3 +152678.368}
SPL {X  -135.604, Y  +763.621, Z    +0.000, E1   -63.883, E3 +152687.970}
SPL {X  -131.007, Y  +770.183, Z    +0.000, E1   -63.497, E3 +152695.256}
SPL {X   -85.750, Y  +811.910, Z    +0.000, E1   -55.921, E3 +152799.208}
ENDSPLINE

SPLINE
SPL {X  -114.463, Y  +789.295, Z    +0.000, E1   -54.865, E3 +152968.475}
SPL {X  -144.553, Y  +748.431, Z    +0.000, E1   -44.979, E3 +152979.183}
SPL {X  -156.024, Y  +720.050, Z    +0.000, E1   -33.178, E3 +152980.750}
SPL {X  -160.714, Y  +699.606, Z    +0.000, E1   -21.520, E3 +152982.624}
SPL {X  -162.196, Y  +687.741, Z    +0.000, E1   -13.310, E3 +152983.151}
SPL {X  -162.791, Y  +676.596, Z    +0.000, E1    -4.586, E3 +152983.435}
SPL {X  -162.820, Y  +671.548, Z    +0.000, E1    -0.068, E3 +152982.912}
SPL {X  -162.820, Y  +669.949, Z    +0.000, E1    +2.213, E3 +152982.600}
SPL {X  -162.820, Y  +664.754, Z    +0.000, E1   +11.697, E3 +152982.499}
SPL {X  -162.820, Y  +658.944, Z    +0.000, E1   +23.544, E3 +152982.667}
SPL {X  -162.820, Y  +650.349, Z    +0.000, E1   +39.427, E3 +152982.164}
SPL {X  -162.820, Y  +632.228, Z    +0.000, E1   +60.508, E3 +152981.394}
SPL {X  -162.820, Y  +572.535, Z    +0.000, E1   +70.270, E3 +153003.439}
SPL {X  -162.820, Y  +446.522, Z    +0.000, E1   +69.253, E3 +153087.263}
SPL {X  -162.820, Y  +440.686, Z    +0.000, E1   +68.127, E3 +153102.138}
SPL {X  -162.820, Y  +421.575, Z    +0.000, E1   +68.212, E3 +153117.201}
SPL {X  -162.820, Y  +409.792, Z    +0.000, E1   +68.121, E3 +153127.792}
SPL {X  -162.820, Y  +394.392, Z    +0.000, E1   +68.165, E3 +153140.367}
SPL {X  -162.820, Y  +385.264, Z    +0.000, E1   +67.766, E3 +153151.282}
ENDSPLINE

SPLINE
SPL {X  -162.820, Y  +397.358, Z    +0.000, E1   +65.083, E3 +153162.284}
ENDSPLINE

SPLINE
SPL {X  -162.719, Y  +374.774, Z    +0.000, E1   +65.968, E3 +153176.768}
SPL {X  -161.214, Y  +357.685, Z    +0.000, E1   +66.686, E3 +153186.523}
SPL {X  -158.043, Y  +341.350, Z    +0.000, E1   +67.216, E3 +153196.632}
SPL {X  -154.848, Y  +330.175, Z    +0.000, E1   +66.891, E3 +153208.443}
SPL {X  -152.657, Y  +323.878, Z    +0.000, E1   +66.551, E3 +153216.178}
SPL {X  -150.291, Y  +317.867, Z    +0.000, E1   +66.312, E3 +153222.954}
SPL {X  -147.540, Y  +311.636, Z    +0.000, E1   +65.718, E3 +153232.223}
SPL {X  -144.094, Y  +304.689, Z    +0.000, E1   +65.338, E3 +153240.437}
SPL {X  -141.093, Y  +299.241, Z    +0.000, E1   +65.039, E3 +153246.750}
SPL {X  -138.425, Y  +294.774, Z    +0.000, E1   +64.416, E3 +153253.934}
SPL {X  -135.581, Y  +290.344, Z    +0.000, E1   +63.996, E3 +153259.766}
SPL {X  -133.378, Y  +287.116, Z    +0.000, E1   +63.482, E3 +153264.930}
SPL {X  -128.896, Y  +281.020, Z    +0.000, E1   +64.005, E3 +153267.699}
SPL {X   -85.291, Y  +241.807, Z    +0.000, E1   +53.957, E3 +153413.107}
ENDSPLINE

